LIN {X 0,Y 536.354,Z 685.03,A -85,B 0,C 180,E1 4123.665,E2 4123.665} C_VEL
LIN {X 0,Y 536.384,Z 685.03,A -85,B 0,C 180,E1 4128.647,E2 4128.647} C_VEL
LIN {X 0,Y 536.412,Z 685.03,A -85,B 0,C 180,E1 4133.543,E2 4133.543} C_VEL
LIN {X 0,Y 536.394,Z 685.03,A -85,B 0,C 180,E1 4138.392,E2 4138.392} C_VEL
LIN {X 0,Y 536.456,Z 685.03,A -85,B 0,C 180,E1 4143.228,E2 4143.228} C_VEL
LIN {X 0,Y 536.326,Z 685.03,A -85,B 0,C 180,E1 4148.09,E2 4148.09} C_VEL
LIN {X 0,Y 536.292,Z 685.03,A -85,B 0,C 180,E1 4153.011,E2 4153.011} C_VEL
LIN {X 0,Y 536.25,Z 685.03,A -85,B 0,C 180,E1 4158.034,E2 4158.034} C_VEL
LIN {X 0,Y 536.123,Z 685.03,A -85,B 0,C 180,E1 4163.209,E2 4163.209} C_VEL
LIN {X 0,Y 536.061,Z 685.03,A -85,B 0,C 180,E1 4166.771,E2 4166.771} C_VEL
LIN {X 0,Y 531.944,Z 685.03,A -85,B 0,C 180,E1 4168.601,E2 4168.601} C_VEL
LIN {X 0,Y 528.057,Z 685.03,A -85,B 0,C 180,E1 4170.459,E2 4170.459} C_VEL
LIN {X 0,Y 528.176,Z 685.03,A -85,B 0,C 180,E1 4176.874,E2 4176.874} C_VEL
LIN {X 0,Y 528.094,Z 685.03,A -85,B 0,C 180,E1 4183.298,E2 4183.298} C_VEL
LIN {X 0,Y 527.996,Z 685.03,A -85,B 0,C 180,E1 4188.904,E2 4188.904} C_VEL
LIN {X 0,Y 528.097,Z 685.034,A -85,B 0,C 180,E1 4193.319,E2 4193.319} C_VEL
LIN {X 0,Y 532.088,Z 694.126,A -85,B 0,C 180,E1 4194.343,E2 4194.343} C_VEL
LIN {X 0,Y 535.905,Z 698.294,A -85,B 0,C 180,E1 4195.482,E2 4195.482} C_VEL
LIN {X 0,Y 536.503,Z 702.972,A -85,B 0,C 180,E1 4195.991,E2 4195.991} C_VEL
LIN {X 0,Y 540.933,Z 714.461,A -85,B 0,C 180,E1 4196.486,E2 4196.486} C_VEL
LIN {X 0,Y 540.144,Z 776.912,A -85,B 0,C 180,E1 4197.563,E2 4197.563} C_VEL
LIN {X 0,Y 538.76,Z 815.29,A -85,B 0,C 180,E1 4198.857,E2 4198.857} C_VEL
LIN {X 0,Y 536.782,Z 852.451,A -85,B 0,C 180,E1 4200.764,E2 4200.764} C_VEL
LIN {X 0,Y 534.633,Z 888.686,A -85,B 0,C 180,E1 4203.381,E2 4203.381} C_VEL
LIN {X 0,Y 532.572,Z 920.102,A -85,B 0,C 180,E1 4206.409,E2 4206.409} C_VEL
LIN {X 0,Y 530.859,Z 948.755,A -85,B 0,C 180,E1 4210.057,E2 4210.057} C_VEL
LIN {X 0,Y 529.67,Z 971.396,A -85,B 0,C 180,E1 4213.874,E2 4213.874} C_VEL
LIN {X 0,Y 529.13,Z 988.021,A -85,B 0,C 180,E1 4217.652,E2 4217.652} C_VEL
LIN {X 0,Y 528.922,Z 999.717,A -85,B 0,C 180,E1 4221.388,E2 4221.388} C_VEL
LIN {X 0,Y 528.766,Z 1006.986,A -85,B 0,C 180,E1 4225.091,E2 4225.091} C_VEL
LIN {X 0,Y 528.757,Z 1010.108,A -85,B 0,C 180,E1 4228.367,E2 4228.367} C_VEL
LIN {X 0,Y 528.747,Z 1009.367,A -85,B 0,C 180,E1 4232.749,E2 4232.749} C_VEL
LIN {X 0,Y 528.862,Z 1004.239,A -85,B 0,C 180,E1 4236.556,E2 4236.556} C_VEL
LIN {X 0,Y 528.962,Z 994.396,A -85,B 0,C 180,E1 4240.488,E2 4240.488} C_VEL
LIN {X 0,Y 529.503,Z 979.171,A -85,B 0,C 180,E1 4244.506,E2 4244.506} C_VEL
LIN {X 0,Y 530.406,Z 958.359,A -85,B 0,C 180,E1 4248.455,E2 4248.455} C_VEL
LIN {X 0,Y 531.902,Z 931.392,A -85,B 0,C 180,E1 4252.271,E2 4252.271} C_VEL
LIN {X 0,Y 533.823,Z 900.632,A -85,B 0,C 180,E1 4255.566,E2 4255.566} C_VEL
LIN {X 0,Y 535.948,Z 866.542,A -85,B 0,C 180,E1 4258.318,E2 4258.318} C_VEL
LIN {X 0,Y 538.081,Z 828.372,A -85,B 0,C 180,E1 4260.553,E2 4260.553} C_VEL
LIN {X 0,Y 539.691,Z 789.324,A -85,B 0,C 180,E1 4262.095,E2 4262.095} C_VEL
LIN {X 0,Y 540.833,Z 748.246,A -85,B 0,C 180,E1 4262.995,E2 4262.995} C_VEL
LIN {X 0,Y 540.481,Z 711.306,A -85,B 0,C 180,E1 4263.595,E2 4263.595} C_VEL
LIN {X 0,Y 535.854,Z 701.121,A -85,B 0,C 180,E1 4264.154,E2 4264.154} C_VEL
LIN {X 0,Y 535.477,Z 697.832,A -85,B 0,C 180,E1 4264.694,E2 4264.694} C_VEL
LIN {X 0,Y 531.547,Z 693.051,A -85,B 0,C 180,E1 4265.81,E2 4265.81} C_VEL
LIN {X 0,Y 528.087,Z 685.03,A -85,B 0,C 180,E1 4266.686,E2 4266.686} C_VEL
LIN {X 0,Y 528.034,Z 685.03,A -85,B 0,C 180,E1 4273.31,E2 4273.31} C_VEL
LIN {X 0,Y 528.107,Z 685.03,A -85,B 0,C 180,E1 4278.913,E2 4278.913} C_VEL
LIN {X 0,Y 528.109,Z 685.03,A -85,B 0,C 180,E1 4285.146,E2 4285.146} C_VEL
LIN {X 0,Y 528.131,Z 685.03,A -85,B 0,C 180,E1 4290.938,E2 4290.938} C_VEL
LIN {X 0,Y 528.203,Z 685.03,A -85,B 0,C 180,E1 4296.422,E2 4296.422} C_VEL
LIN {X 0,Y 528.353,Z 685.03,A -85,B 0,C 180,E1 4302.243,E2 4302.243} C_VEL
LIN {X 0,Y 532.473,Z 702.678,A -85,B 0,C 180,E1 4302.729,E2 4302.729} C_VEL
LIN {X 0,Y 532.139,Z 746.804,A -85,B 0,C 180,E1 4303.524,E2 4303.524} C_VEL
LIN {X 0,Y 531.58,Z 774.498,A -85,B 0,C 180,E1 4304.67,E2 4304.67} C_VEL
LIN {X 0,Y 530.64,Z 800.027,A -85,B 0,C 180,E1 4306.429,E2 4306.429} C_VEL
LIN {X 0,Y 529.919,Z 821.879,A -85,B 0,C 180,E1 4308.72,E2 4308.72} C_VEL
LIN {X 0,Y 529.325,Z 840.1,A -85,B 0,C 180,E1 4311.596,E2 4311.596} C_VEL
LIN {X 0,Y 529.05,Z 851.376,A -85,B 0,C 180,E1 4314.267,E2 4314.267} C_VEL
LIN {X 0,Y 529.003,Z 857.801,A -85,B 0,C 180,E1 4316.844,E2 4316.844} C_VEL
LIN {X 0,Y 528.911,Z 860.413,A -85,B 0,C 180,E1 4319.996,E2 4319.996} C_VEL
LIN {X 0,Y 528.996,Z 857.464,A -85,B 0,C 180,E1 4323.267,E2 4323.267} C_VEL
LIN {X 0,Y 529.045,Z 849.615,A -85,B 0,C 180,E1 4326.136,E2 4326.136} C_VEL
LIN {X 0,Y 529.361,Z 835.063,A -85,B 0,C 180,E1 4329.223,E2 4329.223} C_VEL
LIN {X 0,Y 530.002,Z 817.359,A -85,B 0,C 180,E1 4331.7,E2 4331.7} C_VEL
LIN {X 0,Y 530.789,Z 794.591,A -85,B 0,C 180,E1 4333.874,E2 4333.874} C_VEL
LIN {X 0,Y 531.58,Z 768.365,A -85,B 0,C 180,E1 4335.503,E2 4335.503} C_VEL
LIN {X 0,Y 532.203,Z 738.767,A -85,B 0,C 180,E1 4336.565,E2 4336.565} C_VEL
LIN {X 0,Y 531.65,Z 697.002,A -85,B 0,C 180,E1 4337.27,E2 4337.27} C_VEL
LIN {X 0,Y 528.402,Z 685.03,A -85,B 0,C 180,E1 4337.66,E2 4337.66} C_VEL
LIN {X 0,Y 528.196,Z 685.03,A -85,B 0,C 180,E1 4343.894,E2 4343.894} C_VEL
LIN {X 0,Y 528.104,Z 685.03,A -85,B 0,C 180,E1 4349.055,E2 4349.055} C_VEL
LIN {X 0,Y 528.107,Z 685.03,A -85,B 0,C 180,E1 4354.845,E2 4354.845} C_VEL
LIN {X 0,Y 528.115,Z 685.03,A -85,B 0,C 180,E1 4359.505,E2 4359.505} C_VEL
LIN {X 0,Y 528.084,Z 685.03,A -85,B 0,C 180,E1 4365.582,E2 4365.582} C_VEL
LIN {X 0,Y 528.122,Z 685.03,A -85,B 0,C 180,E1 4371.047,E2 4371.047} C_VEL
LIN {X 0,Y 528.093,Z 685.03,A -85,B 0,C 180,E1 4377.113,E2 4377.113} C_VEL
LIN {X 0,Y 528.209,Z 685.03,A -85,B 0,C 180,E1 4382.796,E2 4382.796} C_VEL
LIN {X 0,Y 528.294,Z 685.296,A -85,B 0,C 180,E1 4386.535,E2 4386.535} C_VEL
LIN {X 0,Y 534.475,Z 708.657,A -85,B 0,C 180,E1 4387.48,E2 4387.48} C_VEL
LIN {X 0,Y 533.347,Z 740.861,A -85,B 0,C 180,E1 4388.886,E2 4388.886} C_VEL
LIN {X 0,Y 531.992,Z 771.472,A -85,B 0,C 180,E1 4390.958,E2 4390.958} C_VEL
LIN {X 0,Y 530.758,Z 798.135,A -85,B 0,C 180,E1 4393.479,E2 4393.479} C_VEL
LIN {X 0,Y 529.823,Z 820.92,A -85,B 0,C 180,E1 4396.46,E2 4396.46} C_VEL
LIN {X 0,Y 529.261,Z 838.534,A -85,B 0,C 180,E1 4399.708,E2 4399.708} C_VEL
LIN {X 0,Y 528.963,Z 850.704,A -85,B 0,C 180,E1 4403.033,E2 4403.033} C_VEL
LIN {X 0,Y 528.87,Z 858.388,A -85,B 0,C 180,E1 4406.726,E2 4406.726} C_VEL
LIN {X 0,Y 528.806,Z 860.497,A -85,B 0,C 180,E1 4409.998,E2 4409.998} C_VEL
LIN {X 0,Y 528.869,Z 858.264,A -85,B 0,C 180,E1 4413.269,E2 4413.269} C_VEL
LIN {X 0,Y 528.989,Z 850.471,A -85,B 0,C 180,E1 4416.961,E2 4416.961} C_VEL
LIN {X 0,Y 529.325,Z 837.086,A -85,B 0,C 180,E1 4420.514,E2 4420.514} C_VEL
LIN {X 0,Y 529.976,Z 817.91,A -85,B 0,C 180,E1 4423.9,E2 4423.9} C_VEL
LIN {X 0,Y 530.907,Z 793.972,A -85,B 0,C 180,E1 4426.887,E2 4426.887} C_VEL
LIN {X 0,Y 532.18,Z 766.335,A -85,B 0,C 180,E1 4429.352,E2 4429.352} C_VEL
LIN {X 0,Y 533.507,Z 736.298,A -85,B 0,C 180,E1 4431.263,E2 4431.263} C_VEL
LIN {X 0,Y 534.003,Z 703.097,A -85,B 0,C 180,E1 4432.636,E2 4432.636} C_VEL
LIN {X 0,Y 528.39,Z 685.03,A -85,B 0,C 180,E1 4433.406,E2 4433.406} C_VEL
LIN {X 0,Y 528.218,Z 685.03,A -85,B 0,C 180,E1 4439.054,E2 4439.054} C_VEL
LIN {X 0,Y 528.144,Z 685.03,A -85,B 0,C 180,E1 4444.849,E2 4444.849} C_VEL
LIN {X 0,Y 527.985,Z 685.03,A -85,B 0,C 180,E1 4451.097,E2 4451.097} C_VEL
LIN {X 0,Y 528.062,Z 685.03,A -85,B 0,C 180,E1 4456.709,E2 4456.709} C_VEL
LIN {X 0,Y 528.163,Z 685.03,A -85,B 0,C 180,E1 4463.128,E2 4463.128} C_VEL
LIN {X 0,Y 528.134,Z 685.03,A -85,B 0,C 180,E1 4469.056,E2 4469.056} C_VEL
LIN {X 0,Y 528.231,Z 685.03,A -85,B 0,C 180,E1 4474.634,E2 4474.634} C_VEL
LIN {X 0,Y 528.453,Z 685.03,A -85,B 0,C 180,E1 4480.445,E2 4480.445} C_VEL
LIN {X 0,Y 528.576,Z 685.03,A -85,B 0,C 180,E1 4486.803,E2 4486.803} C_VEL
LIN {X 0,Y 528.49,Z 685.03,A -85,B 0,C 180,E1 4492.655,E2 4492.655} C_VEL
LIN {X 0,Y 528.516,Z 685.03,A -85,B 0,C 180,E1 4498.368,E2 4498.368} C_VEL
LIN {X 0,Y 528.569,Z 685.03,A -85,B 0,C 180,E1 4503.277,E2 4503.277} C_VEL
LIN {X 0,Y 528.43,Z 685.03,A -85,B 0,C 180,E1 4508.212,E2 4508.212} C_VEL
LIN {X 0,Y 528.339,Z 685.03,A -85,B 0,C 180,E1 4513.811,E2 4513.811} C_VEL
LIN {X 0,Y 528.331,Z 685.03,A -85,B 0,C 180,E1 4519.517,E2 4519.517} C_VEL
LIN {X 0,Y 528.183,Z 685.03,A -85,B 0,C 180,E1 4525.377,E2 4525.377} C_VEL
LIN {X 0,Y 528.057,Z 685.03,A -85,B 0,C 180,E1 4530.459,E2 4530.459} C_VEL
LIN {X 0,Y 525.578,Z 685.03,A -85,B 0,C 180,E1 4531.861,E2 4531.861} C_VEL
LIN {X 0,Y 520.171,Z 685.03,A -85,B 0,C 180,E1 4533.962,E2 4533.962} C_VEL
LIN {X 0,Y 520.069,Z 685.03,A -85,B 0,C 180,E1 4534.205,E2 4534.205} C_VEL
LIN {X 0,Y 520.223,Z 685.03,A -85,B 0,C 180,E1 4539.655,E2 4539.655} C_VEL
LIN {X 0,Y 520.13,Z 685.03,A -85,B 0,C 180,E1 4545.871,E2 4545.871} C_VEL
LIN {X 0,Y 520.099,Z 685.03,A -85,B 0,C 180,E1 4551.57,E2 4551.57} C_VEL
LIN {X 0,Y 520.162,Z 685.3,A -85,B 0,C 180,E1 4552.811,E2 4552.811} C_VEL
LIN {X 0,Y 524.281,Z 695.521,A -85,B 0,C 180,E1 4553.697,E2 4553.697} C_VEL
LIN {X 0,Y 529.992,Z 703.357,A -85,B 0,C 180,E1 4554.791,E2 4554.791} C_VEL
LIN {X 0,Y 531.939,Z 706.912,A -85,B 0,C 180,E1 4555.435,E2 4555.435} C_VEL
LIN {X 0,Y 532.885,Z 711.836,A -85,B 0,C 180,E1 4555.869,E2 4555.869} C_VEL
LIN {X 0,Y 534.317,Z 717.12,A -85,B 0,C 180,E1 4556.057,E2 4556.057} C_VEL
LIN {X 0,Y 533.477,Z 776.899,A -85,B 0,C 180,E1 4557.107,E2 4557.107} C_VEL
LIN {X 0,Y 531.892,Z 815.592,A -85,B 0,C 180,E1 4558.424,E2 4558.424} C_VEL
LIN {X 0,Y 529.702,Z 853.612,A -85,B 0,C 180,E1 4560.413,E2 4560.413} C_VEL
LIN {X 0,Y 527.388,Z 888.681,A -85,B 0,C 180,E1 4562.986,E2 4562.986} C_VEL
LIN {X 0,Y 525.127,Z 920.219,A -85,B 0,C 180,E1 4566.068,E2 4566.068} C_VEL
LIN {X 0,Y 523.234,Z 948.76,A -85,B 0,C 180,E1 4569.754,E2 4569.754} C_VEL
LIN {X 0,Y 521.935,Z 971.4,A -85,B 0,C 180,E1 4573.629,E2 4573.629} C_VEL
LIN {X 0,Y 521.287,Z 988.024,A -85,B 0,C 180,E1 4577.463,E2 4577.463} C_VEL
LIN {X 0,Y 521.052,Z 999.717,A -85,B 0,C 180,E1 4581.257,E2 4581.257} C_VEL
LIN {X 0,Y 520.871,Z 1006.989,A -85,B 0,C 180,E1 4585.016,E2 4585.016} C_VEL
LIN {X 0,Y 520.87,Z 1010.11,A -85,B 0,C 180,E1 4588.342,E2 4588.342} C_VEL
LIN {X 0,Y 520.994,Z 1010.107,A -85,B 0,C 180,E1 4591.662,E2 4591.662} C_VEL
LIN {X 0,Y 520.997,Z 1005.741,A -85,B 0,C 180,E1 4595.821,E2 4595.821} C_VEL
LIN {X 0,Y 521.085,Z 996.126,A -85,B 0,C 180,E1 4600.075,E2 4600.075} C_VEL
LIN {X 0,Y 521.585,Z 981.334,A -85,B 0,C 180,E1 4604.23,E2 4604.23} C_VEL
LIN {X 0,Y 522.578,Z 961.26,A -85,B 0,C 180,E1 4608.245,E2 4608.245} C_VEL
LIN {X 0,Y 524.078,Z 936.283,A -85,B 0,C 180,E1 4611.986,E2 4611.986} C_VEL
LIN {X 0,Y 526.175,Z 905.44,A -85,B 0,C 180,E1 4615.483,E2 4615.483} C_VEL
LIN {X 0,Y 528.495,Z 871.136,A -85,B 0,C 180,E1 4618.404,E2 4618.404} C_VEL
LIN {X 0,Y 530.864,Z 833.862,A -85,B 0,C 180,E1 4620.715,E2 4620.715} C_VEL
LIN {X 0,Y 532.803,Z 795.147,A -85,B 0,C 180,E1 4622.354,E2 4622.354} C_VEL
LIN {X 0,Y 534.124,Z 756.8,A -85,B 0,C 180,E1 4623.314,E2 4623.314} C_VEL
LIN {X 0,Y 533.814,Z 713.846,A -85,B 0,C 180,E1 4624.031,E2 4624.031} C_VEL
LIN {X 0,Y 531.986,Z 709.074,A -85,B 0,C 180,E1 4624.335,E2 4624.335} C_VEL
LIN {X 0,Y 531.319,Z 704.389,A -85,B 0,C 180,E1 4624.917,E2 4624.917} C_VEL
LIN {X 0,Y 526.441,Z 699.138,A -85,B 0,C 180,E1 4625.909,E2 4625.909} C_VEL
LIN {X 0,Y 521.184,Z 689.298,A -85,B 0,C 180,E1 4626.821,E2 4626.821} C_VEL
LIN {X 0,Y 520.132,Z 685.03,A -85,B 0,C 180,E1 4627.142,E2 4627.142} C_VEL
LIN {X 0,Y 520.131,Z 685.03,A -85,B 0,C 180,E1 4633.506,E2 4633.506} C_VEL
LIN {X 0,Y 520.201,Z 685.03,A -85,B 0,C 180,E1 4638.964,E2 4638.964} C_VEL
LIN {X 0,Y 520.165,Z 685.03,A -85,B 0,C 180,E1 4644.534,E2 4644.534} C_VEL
LIN {X 0,Y 520.203,Z 685.03,A -85,B 0,C 180,E1 4650.497,E2 4650.497} C_VEL
LIN {X 0,Y 520.302,Z 685.03,A -85,B 0,C 180,E1 4656.042,E2 4656.042} C_VEL
LIN {X 0,Y 520.458,Z 685.03,A -85,B 0,C 180,E1 4661.896,E2 4661.896} C_VEL
LIN {X 0,Y 525.118,Z 704.487,A -85,B 0,C 180,E1 4662.445,E2 4662.445} C_VEL
LIN {X 0,Y 524.688,Z 748.901,A -85,B 0,C 180,E1 4663.283,E2 4663.283} C_VEL
LIN {X 0,Y 524.081,Z 776.919,A -85,B 0,C 180,E1 4664.484,E2 4664.484} C_VEL
LIN {X 0,Y 523.141,Z 801.802,A -85,B 0,C 180,E1 4666.242,E2 4666.242} C_VEL
LIN {X 0,Y 522.363,Z 823.118,A -85,B 0,C 180,E1 4668.512,E2 4668.512} C_VEL
LIN {X 0,Y 521.688,Z 840.432,A -85,B 0,C 180,E1 4671.262,E2 4671.262} C_VEL
LIN {X 0,Y 521.247,Z 852.269,A -85,B 0,C 180,E1 4674.181,E2 4674.181} C_VEL
LIN {X 0,Y 521.09,Z 859.131,A -85,B 0,C 180,E1 4677.362,E2 4677.362} C_VEL
LIN {X 0,Y 521.032,Z 860.825,A -85,B 0,C 180,E1 4679.996,E2 4679.996} C_VEL
LIN {X 0,Y 521.117,Z 857.949,A -85,B 0,C 180,E1 4683.316,E2 4683.316} C_VEL
LIN {X 0,Y 521.262,Z 848.872,A -85,B 0,C 180,E1 4686.645,E2 4686.645} C_VEL
LIN {X 0,Y 521.691,Z 834.958,A -85,B 0,C 180,E1 4689.569,E2 4689.569} C_VEL
LIN {X 0,Y 522.477,Z 814.795,A -85,B 0,C 180,E1 4692.294,E2 4692.294} C_VEL
LIN {X 0,Y 523.284,Z 791.675,A -85,B 0,C 180,E1 4694.381,E2 4694.381} C_VEL
LIN {X 0,Y 524.182,Z 764.331,A -85,B 0,C 180,E1 4695.974,E2 4695.974} C_VEL
LIN {X 0,Y 524.733,Z 735.414,A -85,B 0,C 180,E1 4696.912,E2 4696.912} C_VEL
LIN {X 0,Y 524.25,Z 698.598,A -85,B 0,C 180,E1 4697.53,E2 4697.53} C_VEL
LIN {X 0,Y 520.493,Z 685.03,A -85,B 0,C 180,E1 4697.928,E2 4697.928} C_VEL
LIN {X 0,Y 520.3,Z 685.03,A -85,B 0,C 180,E1 4703.95,E2 4703.95} C_VEL
LIN {X 0,Y 520.176,Z 685.03,A -85,B 0,C 180,E1 4709.541,E2 4709.541} C_VEL
LIN {X 0,Y 520.204,Z 685.03,A -85,B 0,C 180,E1 4715.678,E2 4715.678} C_VEL
LIN {X 0,Y 520.144,Z 685.03,A -85,B 0,C 180,E1 4721.029,E2 4721.029} C_VEL
LIN {X 0,Y 520.167,Z 685.03,A -85,B 0,C 180,E1 4726.479,E2 4726.479} C_VEL
LIN {X 0,Y 520.207,Z 685.03,A -85,B 0,C 180,E1 4732.466,E2 4732.466} C_VEL
LIN {X 0,Y 520.218,Z 685.03,A -85,B 0,C 180,E1 4738.52,E2 4738.52} C_VEL
LIN {X 0,Y 520.312,Z 685.03,A -85,B 0,C 180,E1 4744.209,E2 4744.209} C_VEL
LIN {X 0,Y 520.395,Z 685.6,A -85,B 0,C 180,E1 4746.14,E2 4746.14} C_VEL
LIN {X 0,Y 527.258,Z 710.651,A -85,B 0,C 180,E1 4747.185,E2 4747.185} C_VEL
LIN {X 0,Y 526.023,Z 743.222,A -85,B 0,C 180,E1 4748.647,E2 4748.647} C_VEL
LIN {X 0,Y 524.583,Z 772.51,A -85,B 0,C 180,E1 4750.679,E2 4750.679} C_VEL
LIN {X 0,Y 523.113,Z 798.31,A -85,B 0,C 180,E1 4753.23,E2 4753.23} C_VEL
LIN {X 0,Y 521.98,Z 822.179,A -85,B 0,C 180,E1 4756.46,E2 4756.46} C_VEL
LIN {X 0,Y 521.407,Z 839.142,A -85,B 0,C 180,E1 4759.687,E2 4759.687} C_VEL
LIN {X 0,Y 521.027,Z 851.834,A -85,B 0,C 180,E1 4763.345,E2 4763.345} C_VEL
LIN {X 0,Y 520.97,Z 858.387,A -85,B 0,C 180,E1 4766.676,E2 4766.676} C_VEL
LIN {X 0,Y 520.91,Z 860.497,A -85,B 0,C 180,E1 4769.997,E2 4769.997} C_VEL
LIN {X 0,Y 520.969,Z 858.265,A -85,B 0,C 180,E1 4773.319,E2 4773.319} C_VEL
LIN {X 0,Y 521.127,Z 850.474,A -85,B 0,C 180,E1 4777.067,E2 4777.067} C_VEL
LIN {X 0,Y 521.439,Z 837.884,A -85,B 0,C 180,E1 4780.499,E2 4780.499} C_VEL
LIN {X 0,Y 522.128,Z 819.589,A -85,B 0,C 180,E1 4783.864,E2 4783.864} C_VEL
LIN {X 0,Y 523.275,Z 794.687,A -85,B 0,C 180,E1 4787.1,E2 4787.1} C_VEL
LIN {X 0,Y 524.821,Z 767.548,A -85,B 0,C 180,E1 4789.635,E2 4789.635} C_VEL
LIN {X 0,Y 526.274,Z 737.203,A -85,B 0,C 180,E1 4791.587,E2 4791.587} C_VEL
LIN {X 0,Y 526.687,Z 704.594,A -85,B 0,C 180,E1 4792.96,E2 4792.96} C_VEL
LIN {X 0,Y 520.413,Z 685.03,A -85,B 0,C 180,E1 4793.815,E2 4793.815} C_VEL
LIN {X 0,Y 520.264,Z 685.03,A -85,B 0,C 180,E1 4799.542,E2 4799.542} C_VEL
LIN {X 0,Y 520.158,Z 685.03,A -85,B 0,C 180,E1 4805.464,E2 4805.464} C_VEL
LIN {X 0,Y 520.075,Z 685.03,A -85,B 0,C 180,E1 4811.862,E2 4811.862} C_VEL
LIN {X 0,Y 520.172,Z 685.03,A -85,B 0,C 180,E1 4818.156,E2 4818.156} C_VEL
LIN {X 0,Y 520.189,Z 685.03,A -85,B 0,C 180,E1 4824.316,E2 4824.316} C_VEL
LIN {X 0,Y 520.227,Z 685.03,A -85,B 0,C 180,E1 4830.482,E2 4830.482} C_VEL
LIN {X 0,Y 520.314,Z 685.03,A -85,B 0,C 180,E1 4836.051,E2 4836.051} C_VEL
LIN {X 0,Y 520.508,Z 685.03,A -85,B 0,C 180,E1 4841.409,E2 4841.409} C_VEL
LIN {X 0,Y 520.681,Z 685.03,A -85,B 0,C 180,E1 4846.599,E2 4846.599} C_VEL
LIN {X 0,Y 520.575,Z 685.03,A -85,B 0,C 180,E1 4852.656,E2 4852.656} C_VEL
LIN {X 0,Y 520.641,Z 685.03,A -85,B 0,C 180,E1 4858.343,E2 4858.343} C_VEL
LIN {X 0,Y 520.664,Z 685.03,A -85,B 0,C 180,E1 4863.326,E2 4863.326} C_VEL
LIN {X 0,Y 520.518,Z 685.03,A -85,B 0,C 180,E1 4868.338,E2 4868.338} C_VEL
LIN {X 0,Y 520.48,Z 685.03,A -85,B 0,C 180,E1 4873.414,E2 4873.414} C_VEL
LIN {X 0,Y 520.416,Z 685.03,A -85,B 0,C 180,E1 4878.602,E2 4878.602} C_VEL
LIN {X 0,Y 520.272,Z 685.03,A -85,B 0,C 180,E1 4883.959,E2 4883.959} C_VEL
LIN {X 0,Y 520.174,Z 685.03,A -85,B 0,C 180,E1 4889.55,E2 4889.55} C_VEL
LIN {X 0,Y 520.069,Z 685.03,A -85,B 0,C 180,E1 4894.205,E2 4894.205} C_VEL
LIN {X 0,Y 516.137,Z 685.03,A -85,B 0,C 180,E1 4896.091,E2 4896.091} C_VEL
LIN {X 0,Y 512.287,Z 685.03,A -85,B 0,C 180,E1 4898.006,E2 4898.006} C_VEL
LIN {X 0,Y 512.255,Z 685.03,A -85,B 0,C 180,E1 4902.652,E2 4902.652} C_VEL
LIN {X 0,Y 512.163,Z 685.03,A -85,B 0,C 180,E1 4907.441,E2 4907.441} C_VEL
LIN {X 0,Y 512.192,Z 685.146,A -85,B 0,C 180,E1 4912.26,E2 4912.26} C_VEL
LIN {X 0,Y 517.631,Z 699.651,A -85,B 0,C 180,E1 4913.517,E2 4913.517} C_VEL
LIN {X 0,Y 524.978,Z 709.353,A -85,B 0,C 180,E1 4914.648,E2 4914.648} C_VEL
LIN {X 0,Y 527.259,Z 714.744,A -85,B 0,C 180,E1 4915.325,E2 4915.325} C_VEL
LIN {X 0,Y 527.77,Z 718.696,A -85,B 0,C 180,E1 4915.603,E2 4915.603} C_VEL
LIN {X 0,Y 526.841,Z 777.247,A -85,B 0,C 180,E1 4916.649,E2 4916.649} C_VEL
LIN {X 0,Y 525.111,Z 815.585,A -85,B 0,C 180,E1 4917.968,E2 4917.968} C_VEL
LIN {X 0,Y 522.754,Z 852.996,A -85,B 0,C 180,E1 4919.938,E2 4919.938} C_VEL
LIN {X 0,Y 520.179,Z 888.679,A -85,B 0,C 180,E1 4922.581,E2 4922.581} C_VEL
LIN {X 0,Y 517.707,Z 920.398,A -85,B 0,C 180,E1 4925.724,E2 4925.724} C_VEL
LIN {X 0,Y 515.594,Z 949.007,A -85,B 0,C 180,E1 4929.478,E2 4929.478} C_VEL
LIN {X 0,Y 514.187,Z 971.403,A -85,B 0,C 180,E1 4933.375,E2 4933.375} C_VEL
LIN {X 0,Y 513.478,Z 988.028,A -85,B 0,C 180,E1 4937.269,E2 4937.269} C_VEL
LIN {X 0,Y 513.156,Z 1000.722,A -85,B 0,C 180,E1 4941.547,E2 4941.547} C_VEL
LIN {X 0,Y 512.979,Z 1006.991,A -85,B 0,C 180,E1 4944.939,E2 4944.939} C_VEL
LIN {X 0,Y 512.993,Z 1010.111,A -85,B 0,C 180,E1 4948.317,E2 4948.317} C_VEL
LIN {X 0,Y 513.109,Z 1010.108,A -85,B 0,C 180,E1 4951.688,E2 4951.688} C_VEL
LIN {X 0,Y 513.102,Z 1005.74,A -85,B 0,C 180,E1 4955.911,E2 4955.911} C_VEL
LIN {X 0,Y 513.214,Z 996.317,A -85,B 0,C 180,E1 4960.164,E2 4960.164} C_VEL
LIN {X 0,Y 513.739,Z 982.207,A -85,B 0,C 180,E1 4964.237,E2 4964.237} C_VEL
LIN {X 0,Y 514.816,Z 962.388,A -85,B 0,C 180,E1 4968.326,E2 4968.326} C_VEL
LIN {X 0,Y 516.523,Z 936.281,A -85,B 0,C 180,E1 4972.325,E2 4972.325} C_VEL
LIN {X 0,Y 518.822,Z 905.439,A -85,B 0,C 180,E1 4975.871,E2 4975.871} C_VEL
LIN {X 0,Y 521.365,Z 871.904,A -85,B 0,C 180,E1 4978.767,E2 4978.767} C_VEL
LIN {X 0,Y 523.942,Z 834.623,A -85,B 0,C 180,E1 4981.122,E2 4981.122} C_VEL
LIN {X 0,Y 526.056,Z 795.898,A -85,B 0,C 180,E1 4982.793,E2 4982.793} C_VEL
LIN {X 0,Y 527.517,Z 757.791,A -85,B 0,C 180,E1 4983.769,E2 4983.769} C_VEL
LIN {X 0,Y 527.562,Z 716.814,A -85,B 0,C 180,E1 4984.456,E2 4984.456} C_VEL
LIN {X 0,Y 526.094,Z 710.29,A -85,B 0,C 180,E1 4985.167,E2 4985.167} C_VEL
LIN {X 0,Y 519.052,Z 701.862,A -85,B 0,C 180,E1 4986.228,E2 4986.228} C_VEL
LIN {X 0,Y 513.064,Z 689.146,A -85,B 0,C 180,E1 4987.202,E2 4987.202} C_VEL
LIN {X 0,Y 512.175,Z 685.03,A -85,B 0,C 180,E1 4987.553,E2 4987.553} C_VEL
LIN {X 0,Y 512.187,Z 685.03,A -85,B 0,C 180,E1 4992.665,E2 4992.665} C_VEL
LIN {X 0,Y 512.26,Z 685.03,A -85,B 0,C 180,E1 4997.436,E2 4997.436} C_VEL
LIN {X 0,Y 512.269,Z 685.03,A -85,B 0,C 180,E1 5002.696,E2 5002.696} C_VEL
LIN {X 0,Y 512.257,Z 685.03,A -85,B 0,C 180,E1 5008.69,E2 5008.69} C_VEL
LIN {X 0,Y 512.327,Z 685.03,A -85,B 0,C 180,E1 5013.779,E2 5013.779} C_VEL
LIN {X 0,Y 512.462,Z 685.03,A -85,B 0,C 180,E1 5019.305,E2 5019.305} C_VEL
LIN {X 0,Y 512.549,Z 685.552,A -85,B 0,C 180,E1 5021.537,E2 5021.537} C_VEL
LIN {X 0,Y 517.769,Z 703.512,A -85,B 0,C 180,E1 5022.11,E2 5022.11} C_VEL
LIN {X 0,Y 517.288,Z 750.923,A -85,B 0,C 180,E1 5023.037,E2 5023.037} C_VEL
LIN {X 0,Y 516.669,Z 778,A -85,B 0,C 180,E1 5024.216,E2 5024.216} C_VEL
LIN {X 0,Y 515.642,Z 803.277,A -85,B 0,C 180,E1 5026.026,E2 5026.026} C_VEL
LIN {X 0,Y 514.745,Z 825.334,A -85,B 0,C 180,E1 5028.429,E2 5028.429} C_VEL
LIN {X 0,Y 513.975,Z 843.001,A -85,B 0,C 180,E1 5031.343,E2 5031.343} C_VEL
LIN {X 0,Y 513.471,Z 854.905,A -85,B 0,C 180,E1 5034.516,E2 5034.516} C_VEL
LIN {X 0,Y 513.333,Z 860.727,A -85,B 0,C 180,E1 5037.469,E2 5037.469} C_VEL
LIN {X 0,Y 513.282,Z 862.188,A -85,B 0,C 180,E1 5039.996,E2 5039.996} C_VEL
LIN {X 0,Y 513.352,Z 859.214,A -85,B 0,C 180,E1 5043.366,E2 5043.366} C_VEL
LIN {X 0,Y 513.51,Z 850.089,A -85,B 0,C 180,E1 5046.746,E2 5046.746} C_VEL
LIN {X 0,Y 513.996,Z 836.089,A -85,B 0,C 180,E1 5049.714,E2 5049.714} C_VEL
LIN {X 0,Y 514.857,Z 815.868,A -85,B 0,C 180,E1 5052.478,E2 5052.478} C_VEL
LIN {X 0,Y 515.729,Z 792.128,A -85,B 0,C 180,E1 5054.64,E2 5054.64} C_VEL
LIN {X 0,Y 516.695,Z 764.192,A -85,B 0,C 180,E1 5056.266,E2 5056.266} C_VEL
LIN {X 0,Y 517.273,Z 734.612,A -85,B 0,C 180,E1 5057.205,E2 5057.205} C_VEL
LIN {X 0,Y 516.63,Z 699.556,A -85,B 0,C 180,E1 5057.803,E2 5057.803} C_VEL
LIN {X 0,Y 512.554,Z 685.03,A -85,B 0,C 180,E1 5058.248,E2 5058.248} C_VEL
LIN {X 0,Y 512.359,Z 685.03,A -85,B 0,C 180,E1 5064.345,E2 5064.345} C_VEL
LIN {X 0,Y 512.213,Z 685.03,A -85,B 0,C 180,E1 5070.048,E2 5070.048} C_VEL
LIN {X 0,Y 512.286,Z 685.03,A -85,B 0,C 180,E1 5076.087,E2 5076.087} C_VEL
LIN {X 0,Y 512.257,Z 685.03,A -85,B 0,C 180,E1 5080.387,E2 5080.387} C_VEL
LIN {X 0,Y 512.206,Z 685.03,A -85,B 0,C 180,E1 5084.997,E2 5084.997} C_VEL
LIN {X 0,Y 512.288,Z 685.03,A -85,B 0,C 180,E1 5089.972,E2 5089.972} C_VEL
LIN {X 0,Y 512.194,Z 685.03,A -85,B 0,C 180,E1 5095.955,E2 5095.955} C_VEL
LIN {X 0,Y 512.36,Z 685.03,A -85,B 0,C 180,E1 5102.057,E2 5102.057} C_VEL
LIN {X 0,Y 512.427,Z 685.062,A -85,B 0,C 180,E1 5105.711,E2 5105.711} C_VEL
LIN {X 0,Y 520.066,Z 712.731,A -85,B 0,C 180,E1 5106.885,E2 5106.885} C_VEL
LIN {X 0,Y 518.771,Z 744.492,A -85,B 0,C 180,E1 5108.337,E2 5108.337} C_VEL
LIN {X 0,Y 517.221,Z 773.73,A -85,B 0,C 180,E1 5110.392,E2 5110.392} C_VEL
LIN {X 0,Y 515.627,Z 799.545,A -85,B 0,C 180,E1 5112.98,E2 5112.98} C_VEL
LIN {X 0,Y 514.318,Z 822.023,A -85,B 0,C 180,E1 5116.151,E2 5116.151} C_VEL
LIN {X 0,Y 513.471,Z 840.437,A -85,B 0,C 180,E1 5119.841,E2 5119.841} C_VEL
LIN {X 0,Y 513.165,Z 851.831,A -85,B 0,C 180,E1 5123.242,E2 5123.242} C_VEL
LIN {X 0,Y 513.081,Z 858.387,A -85,B 0,C 180,E1 5126.625,E2 5126.625} C_VEL
LIN {X 0,Y 512.993,Z 860.423,A -85,B 0,C 180,E1 5130.376,E2 5130.376} C_VEL
LIN {X 0,Y 513.103,Z 857.062,A -85,B 0,C 180,E1 5134.214,E2 5134.214} C_VEL
LIN {X 0,Y 513.335,Z 847.901,A -85,B 0,C 180,E1 5138.024,E2 5138.024} C_VEL
LIN {X 0,Y 513.801,Z 833.266,A -85,B 0,C 180,E1 5141.647,E2 5141.647} C_VEL
LIN {X 0,Y 514.819,Z 813.602,A -85,B 0,C 180,E1 5145.081,E2 5145.081} C_VEL
LIN {X 0,Y 516.236,Z 789.868,A -85,B 0,C 180,E1 5148.011,E2 5148.011} C_VEL
LIN {X 0,Y 517.896,Z 761.609,A -85,B 0,C 180,E1 5150.464,E2 5150.464} C_VEL
LIN {X 0,Y 519.3,Z 731.077,A -85,B 0,C 180,E1 5152.274,E2 5152.274} C_VEL
LIN {X 0,Y 519.362,Z 706.232,A -85,B 0,C 180,E1 5153.289,E2 5153.289} C_VEL
LIN {X 0,Y 512.459,Z 685.03,A -85,B 0,C 180,E1 5154.256,E2 5154.256} C_VEL
LIN {X 0,Y 512.3,Z 685.03,A -85,B 0,C 180,E1 5160.048,E2 5160.048} C_VEL
LIN {X 0,Y 512.201,Z 685.03,A -85,B 0,C 180,E1 5166.101,E2 5166.101} C_VEL
LIN {X 0,Y 512.178,Z 685.03,A -85,B 0,C 180,E1 5170.403,E2 5170.403} C_VEL
LIN {X 0,Y 512.173,Z 685.03,A -85,B 0,C 180,E1 5175.01,E2 5175.01} C_VEL
LIN {X 0,Y 512.296,Z 685.03,A -85,B 0,C 180,E1 5179.982,E2 5179.982} C_VEL
LIN {X 0,Y 512.232,Z 685.03,A -85,B 0,C 180,E1 5185.971,E2 5185.971} C_VEL
LIN {X 0,Y 512.328,Z 685.03,A -85,B 0,C 180,E1 5192.082,E2 5192.082} C_VEL
LIN {X 0,Y 512.428,Z 685.03,A -85,B 0,C 180,E1 5197.497,E2 5197.497} C_VEL
LIN {X 0,Y 512.639,Z 685.03,A -85,B 0,C 180,E1 5202.886,E2 5202.886} C_VEL
LIN {X 0,Y 512.668,Z 685.03,A -85,B 0,C 180,E1 5208.114,E2 5208.114} C_VEL
LIN {X 0,Y 512.705,Z 685.03,A -85,B 0,C 180,E1 5213.243,E2 5213.243} C_VEL
LIN {X 0,Y 512.741,Z 685.03,A -85,B 0,C 180,E1 5218.317,E2 5218.317} C_VEL
LIN {X 0,Y 512.769,Z 685.03,A -85,B 0,C 180,E1 5223.378,E2 5223.378} C_VEL
LIN {X 0,Y 512.611,Z 685.03,A -85,B 0,C 180,E1 5228.467,E2 5228.467} C_VEL
LIN {X 0,Y 512.542,Z 685.03,A -85,B 0,C 180,E1 5233.693,E2 5233.693} C_VEL
LIN {X 0,Y 512.469,Z 685.03,A -85,B 0,C 180,E1 5239.564,E2 5239.564} C_VEL
LIN {X 0,Y 512.335,Z 685.03,A -85,B 0,C 180,E1 5244.354,E2 5244.354} C_VEL
LIN {X 0,Y 512.211,Z 685.03,A -85,B 0,C 180,E1 5250.056,E2 5250.056} C_VEL
LIN {X 0,Y 512.251,Z 685.03,A -85,B 0,C 180,E1 5256.099,E2 5256.099} C_VEL
LIN {X 0,Y 512.287,Z 685.03,A -85,B 0,C 180,E1 5258.006,E2 5258.006} C_VEL
LIN {X 0,Y 509.808,Z 685.03,A -85,B 0,C 180,E1 5259.436,E2 5259.436} C_VEL
LIN {X 0,Y 504.243,Z 685.03,A -85,B 0,C 180,E1 5261.826,E2 5261.826} C_VEL
LIN {X 0,Y 504.187,Z 685.03,A -85,B 0,C 180,E1 5266.499,E2 5266.499} C_VEL
LIN {X 0,Y 504.322,Z 685.713,A -85,B 0,C 180,E1 5271.742,E2 5271.742} C_VEL
LIN {X 0,Y 511.317,Z 704.209,A -85,B 0,C 180,E1 5273.381,E2 5273.381} C_VEL
LIN {X 0,Y 521.17,Z 717.935,A -85,B 0,C 180,E1 5274.88,E2 5274.88} C_VEL
LIN {X 0,Y 521.178,Z 724.456,A -85,B 0,C 180,E1 5275.2,E2 5275.2} C_VEL
LIN {X 0,Y 520.179,Z 778.605,A -85,B 0,C 180,E1 5276.204,E2 5276.204} C_VEL
LIN {X 0,Y 518.33,Z 816.283,A -85,B 0,C 180,E1 5277.532,E2 5277.532} C_VEL
LIN {X 0,Y 515.728,Z 854.016,A -85,B 0,C 180,E1 5279.556,E2 5279.556} C_VEL
LIN {X 0,Y 512.883,Z 889.667,A -85,B 0,C 180,E1 5282.249,E2 5282.249} C_VEL
LIN {X 0,Y 510.163,Z 922.025,A -85,B 0,C 180,E1 5285.539,E2 5285.539} C_VEL
LIN {X 0,Y 507.905,Z 950.005,A -85,B 0,C 180,E1 5289.31,E2 5289.31} C_VEL
LIN {X 0,Y 506.363,Z 972.478,A -85,B 0,C 180,E1 5293.333,E2 5293.333} C_VEL
LIN {X 0,Y 505.56,Z 989.569,A -85,B 0,C 180,E1 5297.504,E2 5297.504} C_VEL
LIN {X 0,Y 505.264,Z 1000.725,A -85,B 0,C 180,E1 5301.414,E2 5301.414} C_VEL
LIN {X 0,Y 505.087,Z 1006.994,A -85,B 0,C 180,E1 5304.86,E2 5304.86} C_VEL
LIN {X 0,Y 505.09,Z 1010.112,A -85,B 0,C 180,E1 5308.291,E2 5308.291} C_VEL
LIN {X 0,Y 505.202,Z 1010.11,A -85,B 0,C 180,E1 5311.714,E2 5311.714} C_VEL
LIN {X 0,Y 505.211,Z 1005.739,A -85,B 0,C 180,E1 5316.004,E2 5316.004} C_VEL
LIN {X 0,Y 505.331,Z 996.316,A -85,B 0,C 180,E1 5320.325,E2 5320.325} C_VEL
LIN {X 0,Y 505.99,Z 981.087,A -85,B 0,C 180,E1 5324.737,E2 5324.737} C_VEL
LIN {X 0,Y 507.172,Z 960.892,A -85,B 0,C 180,E1 5328.885,E2 5328.885} C_VEL
LIN {X 0,Y 509.119,Z 934.459,A -85,B 0,C 180,E1 5332.916,E2 5332.916} C_VEL
LIN {X 0,Y 511.756,Z 903.197,A -85,B 0,C 180,E1 5336.491,E2 5336.491} C_VEL
LIN {X 0,Y 514.52,Z 868.916,A -85,B 0,C 180,E1 5339.427,E2 5339.427} C_VEL
LIN {X 0,Y 517.352,Z 831.713,A -85,B 0,C 180,E1 5341.734,E2 5341.734} C_VEL
LIN {X 0,Y 519.544,Z 792.025,A -85,B 0,C 180,E1 5343.405,E2 5343.405} C_VEL
LIN {X 0,Y 521.064,Z 750.75,A -85,B 0,C 180,E1 5344.377,E2 5344.377} C_VEL
LIN {X 0,Y 521.662,Z 719.901,A -85,B 0,C 180,E1 5344.943,E2 5344.943} C_VEL
LIN {X 0,Y 520.263,Z 715.673,A -85,B 0,C 180,E1 5345.338,E2 5345.338} C_VEL
LIN {X 0,Y 509.915,Z 702.399,A -85,B 0,C 180,E1 5346.61,E2 5346.61} C_VEL
LIN {X 0,Y 504.279,Z 685.03,A -85,B 0,C 180,E1 5347.87,E2 5347.87} C_VEL
LIN {X 0,Y 504.238,Z 685.03,A -85,B 0,C 180,E1 5354.091,E2 5354.091} C_VEL
LIN {X 0,Y 504.299,Z 685.03,A -85,B 0,C 180,E1 5358.829,E2 5358.829} C_VEL
LIN {X 0,Y 504.375,Z 685.03,A -85,B 0,C 180,E1 5363.889,E2 5363.889} C_VEL
LIN {X 0,Y 504.304,Z 685.03,A -85,B 0,C 180,E1 5370.209,E2 5370.209} C_VEL
LIN {X 0,Y 504.413,Z 685.03,A -85,B 0,C 180,E1 5375.238,E2 5375.238} C_VEL
LIN {X 0,Y 504.575,Z 685.031,A -85,B 0,C 180,E1 5381.118,E2 5381.118} C_VEL
LIN {X 0,Y 510.438,Z 706.142,A -85,B 0,C 180,E1 5381.824,E2 5381.824} C_VEL
LIN {X 0,Y 509.868,Z 752.872,A -85,B 0,C 180,E1 5382.783,E2 5382.783} C_VEL
LIN {X 0,Y 509.221,Z 779.689,A -85,B 0,C 180,E1 5383.978,E2 5383.978} C_VEL
LIN {X 0,Y 508.191,Z 803.574,A -85,B 0,C 180,E1 5385.696,E2 5385.696} C_VEL
LIN {X 0,Y 507.278,Z 824.775,A -85,B 0,C 180,E1 5387.979,E2 5387.979} C_VEL
LIN {X 0,Y 506.431,Z 842.357,A -85,B 0,C 180,E1 5390.781,E2 5390.781} C_VEL
LIN {X 0,Y 505.804,Z 855.149,A -85,B 0,C 180,E1 5394.003,E2 5394.003} C_VEL
LIN {X 0,Y 505.589,Z 862.124,A -85,B 0,C 180,E1 5397.43,E2 5397.43} C_VEL
LIN {X 0,Y 505.528,Z 863.551,A -85,B 0,C 180,E1 5399.996,E2 5399.996} C_VEL
LIN {X 0,Y 505.595,Z 860.478,A -85,B 0,C 180,E1 5403.418,E2 5403.418} C_VEL
LIN {X 0,Y 505.77,Z 851.305,A -85,B 0,C 180,E1 5406.85,E2 5406.85} C_VEL
LIN {X 0,Y 506.294,Z 837.22,A -85,B 0,C 180,E1 5409.863,E2 5409.863} C_VEL
LIN {X 0,Y 507.159,Z 818.821,A -85,B 0,C 180,E1 5412.453,E2 5412.453} C_VEL
LIN {X 0,Y 508.132,Z 795.272,A -85,B 0,C 180,E1 5414.703,E2 5414.703} C_VEL
LIN {X 0,Y 509.086,Z 768.748,A -85,B 0,C 180,E1 5416.35,E2 5416.35} C_VEL
LIN {X 0,Y 509.751,Z 739.215,A -85,B 0,C 180,E1 5417.393,E2 5417.393} C_VEL
LIN {X 0,Y 509.252,Z 701.263,A -85,B 0,C 180,E1 5418.064,E2 5418.064} C_VEL
LIN {X 0,Y 504.625,Z 685.03,A -85,B 0,C 180,E1 5418.595,E2 5418.595} C_VEL
LIN {X 0,Y 504.401,Z 685.03,A -85,B 0,C 180,E1 5424.754,E2 5424.754} C_VEL
LIN {X 0,Y 504.303,Z 685.03,A -85,B 0,C 180,E1 5430.569,E2 5430.569} C_VEL
LIN {X 0,Y 504.408,Z 685.03,A -85,B 0,C 180,E1 5436.742,E2 5436.742} C_VEL
LIN {X 0,Y 504.225,Z 685.03,A -85,B 0,C 180,E1 5441.56,E2 5441.56} C_VEL
LIN {X 0,Y 504.229,Z 685.03,A -85,B 0,C 180,E1 5446.496,E2 5446.496} C_VEL
LIN {X 0,Y 504.367,Z 685.03,A -85,B 0,C 180,E1 5453.241,E2 5453.241} C_VEL
LIN {X 0,Y 504.38,Z 685.03,A -85,B 0,C 180,E1 5459.424,E2 5459.424} C_VEL
LIN {X 0,Y 504.485,Z 685.03,A -85,B 0,C 180,E1 5465.276,E2 5465.276} C_VEL
LIN {X 0,Y 512.906,Z 713.471,A -85,B 0,C 180,E1 5466.528,E2 5466.528} C_VEL
LIN {X 0,Y 511.563,Z 745.118,A -85,B 0,C 180,E1 5467.981,E2 5467.981} C_VEL
LIN {X 0,Y 509.902,Z 774.942,A -85,B 0,C 180,E1 5470.099,E2 5470.099} C_VEL
LIN {X 0,Y 508.154,Z 800.777,A -85,B 0,C 180,E1 5472.721,E2 5472.721} C_VEL
LIN {X 0,Y 506.803,Z 822.317,A -85,B 0,C 180,E1 5475.774,E2 5475.774} C_VEL
LIN {X 0,Y 505.814,Z 839.52,A -85,B 0,C 180,E1 5479.251,E2 5479.251} C_VEL
LIN {X 0,Y 505.411,Z 850.918,A -85,B 0,C 180,E1 5482.707,E2 5482.707} C_VEL
LIN {X 0,Y 505.18,Z 858.386,A -85,B 0,C 180,E1 5486.572,E2 5486.572} C_VEL
LIN {X 0,Y 505.16,Z 860.498,A -85,B 0,C 180,E1 5489.997,E2 5489.997} C_VEL
LIN {X 0,Y 505.179,Z 858.267,A -85,B 0,C 180,E1 5493.423,E2 5493.423} C_VEL
LIN {X 0,Y 505.481,Z 849.519,A -85,B 0,C 180,E1 5497.718,E2 5497.718} C_VEL
LIN {X 0,Y 506.083,Z 835.436,A -85,B 0,C 180,E1 5501.609,E2 5501.609} C_VEL
LIN {X 0,Y 507.183,Z 816.554,A -85,B 0,C 180,E1 5505.059,E2 5505.059} C_VEL
LIN {X 0,Y 508.738,Z 792.295,A -85,B 0,C 180,E1 5508.153,E2 5508.153} C_VEL
LIN {X 0,Y 510.527,Z 764.288,A -85,B 0,C 180,E1 5510.66,E2 5510.66} C_VEL
LIN {X 0,Y 512.04,Z 733.931,A -85,B 0,C 180,E1 5512.525,E2 5512.525} C_VEL
LIN {X 0,Y 512.212,Z 708.406,A -85,B 0,C 180,E1 5513.602,E2 5513.602} C_VEL
LIN {X 0,Y 504.478,Z 685.03,A -85,B 0,C 180,E1 5514.682,E2 5514.682} C_VEL
LIN {X 0,Y 504.388,Z 685.03,A -85,B 0,C 180,E1 5520.569,E2 5520.569} C_VEL
LIN {X 0,Y 504.274,Z 685.03,A -85,B 0,C 180,E1 5526.76,E2 5526.76} C_VEL
LIN {X 0,Y 504.151,Z 685.03,A -85,B 0,C 180,E1 5533.505,E2 5533.505} C_VEL
LIN {X 0,Y 504.277,Z 685.03,A -85,B 0,C 180,E1 5538.837,E2 5538.837} C_VEL
LIN {X 0,Y 504.319,Z 685.03,A -85,B 0,C 180,E1 5545.362,E2 5545.362} C_VEL
LIN {X 0,Y 504.354,Z 685.03,A -85,B 0,C 180,E1 5551.406,E2 5551.406} C_VEL
LIN {X 0,Y 504.487,Z 685.03,A -85,B 0,C 180,E1 5557.123,E2 5557.123} C_VEL
LIN {X 0,Y 504.745,Z 685.03,A -85,B 0,C 180,E1 5563.075,E2 5563.075} C_VEL
LIN {X 0,Y 504.758,Z 685.03,A -85,B 0,C 180,E1 5567.925,E2 5567.925} C_VEL
LIN {X 0,Y 504.794,Z 685.03,A -85,B 0,C 180,E1 5573.137,E2 5573.137} C_VEL
LIN {X 0,Y 504.84,Z 685.03,A -85,B 0,C 180,E1 5578.291,E2 5578.291} C_VEL
LIN {X 0,Y 504.863,Z 685.03,A -85,B 0,C 180,E1 5583.431,E2 5583.431} C_VEL
LIN {X 0,Y 504.686,Z 685.03,A -85,B 0,C 180,E1 5589.355,E2 5589.355} C_VEL
LIN {X 0,Y 504.588,Z 685.03,A -85,B 0,C 180,E1 5595.616,E2 5595.616} C_VEL
LIN {X 0,Y 504.518,Z 685.03,A -85,B 0,C 180,E1 5601.036,E2 5601.036} C_VEL
LIN {X 0,Y 504.35,Z 685.03,A -85,B 0,C 180,E1 5606.668,E2 5606.668} C_VEL
LIN {X 0,Y 504.237,Z 685.03,A -85,B 0,C 180,E1 5613.077,E2 5613.077} C_VEL
LIN {X 0,Y 504.356,Z 685.03,A -85,B 0,C 180,E1 5618.931,E2 5618.931} C_VEL
LIN {X 0,Y 504.243,Z 685.03,A -85,B 0,C 180,E1 5621.826,E2 5621.826} C_VEL
LIN {X 0,Y 500.28,Z 685.03,A -85,B 0,C 180,E1 5623.774,E2 5623.774} C_VEL
LIN {X 0,Y 496.305,Z 685.03,A -85,B 0,C 180,E1 5625.753,E2 5625.753} C_VEL
LIN {X 0,Y 496.364,Z 685.177,A -85,B 0,C 180,E1 5631.126,E2 5631.126} C_VEL
LIN {X 0,Y 504.828,Z 708.453,A -85,B 0,C 180,E1 5633.21,E2 5633.21} C_VEL
LIN {X 0,Y 514.564,Z 722.331,A -85,B 0,C 180,E1 5634.696,E2 5634.696} C_VEL
LIN {X 0,Y 513.65,Z 777.212,A -85,B 0,C 180,E1 5635.677,E2 5635.677} C_VEL
LIN {X 0,Y 511.692,Z 815.094,A -85,B 0,C 180,E1 5636.999,E2 5636.999} C_VEL
LIN {X 0,Y 508.827,Z 853.526,A -85,B 0,C 180,E1 5639.064,E2 5639.064} C_VEL
LIN {X 0,Y 505.751,Z 889.255,A -85,B 0,C 180,E1 5641.784,E2 5641.784} C_VEL
LIN {X 0,Y 502.788,Z 922.029,A -85,B 0,C 180,E1 5645.156,E2 5645.156} C_VEL
LIN {X 0,Y 500.359,Z 949.792,A -85,B 0,C 180,E1 5648.949,E2 5648.949} C_VEL
LIN {X 0,Y 498.641,Z 972.477,A -85,B 0,C 180,E1 5653.068,E2 5653.068} C_VEL
LIN {X 0,Y 497.733,Z 989.57,A -85,B 0,C 180,E1 5657.305,E2 5657.305} C_VEL
LIN {X 0,Y 497.389,Z 1000.725,A -85,B 0,C 180,E1 5661.277,E2 5661.277} C_VEL
LIN {X 0,Y 497.195,Z 1006.996,A -85,B 0,C 180,E1 5664.778,E2 5664.778} C_VEL
LIN {X 0,Y 497.213,Z 1010.112,A -85,B 0,C 180,E1 5668.263,E2 5668.263} C_VEL
LIN {X 0,Y 497.298,Z 1010.11,A -85,B 0,C 180,E1 5671.742,E2 5671.742} C_VEL
LIN {X 0,Y 497.334,Z 1005.738,A -85,B 0,C 180,E1 5676.099,E2 5676.099} C_VEL
LIN {X 0,Y 497.449,Z 996.315,A -85,B 0,C 180,E1 5680.49,E2 5680.49} C_VEL
LIN {X 0,Y 498.158,Z 981.658,A -85,B 0,C 180,E1 5684.834,E2 5684.834} C_VEL
LIN {X 0,Y 499.493,Z 960.905,A -85,B 0,C 180,E1 5689.184,E2 5689.184} C_VEL
LIN {X 0,Y 501.655,Z 934.457,A -85,B 0,C 180,E1 5693.277,E2 5693.277} C_VEL
LIN {X 0,Y 504.456,Z 903.417,A -85,B 0,C 180,E1 5696.882,E2 5696.882} C_VEL
LIN {X 0,Y 507.522,Z 868.916,A -85,B 0,C 180,E1 5699.874,E2 5699.874} C_VEL
LIN {X 0,Y 510.551,Z 831.72,A -85,B 0,C 180,E1 5702.208,E2 5702.208} C_VEL
LIN {X 0,Y 512.894,Z 792.59,A -85,B 0,C 180,E1 5703.874,E2 5703.874} C_VEL
LIN {X 0,Y 514.461,Z 753.852,A -85,B 0,C 180,E1 5704.807,E2 5704.807} C_VEL
LIN {X 0,Y 514.454,Z 721.412,A -85,B 0,C 180,E1 5705.351,E2 5705.351} C_VEL
LIN {X 0,Y 501.694,Z 703.599,A -85,B 0,C 180,E1 5706.924,E2 5706.924} C_VEL
LIN {X 0,Y 496.35,Z 685.03,A -85,B 0,C 180,E1 5708.264,E2 5708.264} C_VEL
LIN {X 0,Y 496.333,Z 685.03,A -85,B 0,C 180,E1 5714.375,E2 5714.375} C_VEL
LIN {X 0,Y 496.36,Z 685.03,A -85,B 0,C 180,E1 5720.324,E2 5720.324} C_VEL
LIN {X 0,Y 496.357,Z 685.03,A -85,B 0,C 180,E1 5726.822,E2 5726.822} C_VEL
LIN {X 0,Y 496.42,Z 685.03,A -85,B 0,C 180,E1 5732.871,E2 5732.871} C_VEL
LIN {X 0,Y 496.589,Z 685.03,A -85,B 0,C 180,E1 5738.612,E2 5738.612} C_VEL
LIN {X 0,Y 496.671,Z 685.03,A -85,B 0,C 180,E1 5740.677,E2 5740.677} C_VEL
LIN {X 0,Y 503.146,Z 707.225,A -85,B 0,C 180,E1 5741.498,E2 5741.498} C_VEL
LIN {X 0,Y 502.474,Z 754.895,A -85,B 0,C 180,E1 5742.521,E2 5742.521} C_VEL
LIN {X 0,Y 501.789,Z 781.42,A -85,B 0,C 180,E1 5743.734,E2 5743.734} C_VEL
LIN {X 0,Y 500.667,Z 806.81,A -85,B 0,C 180,E1 5745.632,E2 5745.632} C_VEL
LIN {X 0,Y 499.637,Z 827.932,A -85,B 0,C 180,E1 5748.013,E2 5748.013} C_VEL
LIN {X 0,Y 498.72,Z 844.97,A -85,B 0,C 180,E1 5750.862,E2 5750.862} C_VEL
LIN {X 0,Y 498.105,Z 856.584,A -85,B 0,C 180,E1 5753.91,E2 5753.91} C_VEL
LIN {X 0,Y 497.883,Z 862.366,A -85,B 0,C 180,E1 5756.521,E2 5756.521} C_VEL
LIN {X 0,Y 497.779,Z 864.914,A -85,B 0,C 180,E1 5759.996,E2 5759.996} C_VEL
LIN {X 0,Y 497.814,Z 861.745,A -85,B 0,C 180,E1 5763.472,E2 5763.472} C_VEL
LIN {X 0,Y 498.023,Z 852.522,A -85,B 0,C 180,E1 5766.957,E2 5766.957} C_VEL
LIN {X 0,Y 498.576,Z 838.59,A -85,B 0,C 180,E1 5769.977,E2 5769.977} C_VEL
LIN {X 0,Y 499.517,Z 819.897,A -85,B 0,C 180,E1 5772.646,E2 5772.646} C_VEL
LIN {X 0,Y 500.57,Z 795.855,A -85,B 0,C 180,E1 5774.967,E2 5774.967} C_VEL
LIN {X 0,Y 501.608,Z 768.634,A -85,B 0,C 180,E1 5776.657,E2 5776.657} C_VEL
LIN {X 0,Y 502.268,Z 740.39,A -85,B 0,C 180,E1 5777.66,E2 5777.66} C_VEL
LIN {X 0,Y 501.815,Z 702.718,A -85,B 0,C 180,E1 5778.342,E2 5778.342} C_VEL
LIN {X 0,Y 496.715,Z 685.03,A -85,B 0,C 180,E1 5778.942,E2 5778.942} C_VEL
LIN {X 0,Y 496.498,Z 685.03,A -85,B 0,C 180,E1 5785.176,E2 5785.176} C_VEL
LIN {X 0,Y 496.3,Z 685.03,A -85,B 0,C 180,E1 5791.632,E2 5791.632} C_VEL
LIN {X 0,Y 496.431,Z 685.03,A -85,B 0,C 180,E1 5797.776,E2 5797.776} C_VEL
LIN {X 0,Y 496.313,Z 685.03,A -85,B 0,C 180,E1 5804.36,E2 5804.36} C_VEL
LIN {X 0,Y 496.373,Z 685.03,A -85,B 0,C 180,E1 5810.321,E2 5810.321} C_VEL
LIN {X 0,Y 496.359,Z 685.03,A -85,B 0,C 180,E1 5816.818,E2 5816.818} C_VEL
LIN {X 0,Y 496.478,Z 685.03,A -85,B 0,C 180,E1 5822.872,E2 5822.872} C_VEL
LIN {X 0,Y 496.583,Z 685.733,A -85,B 0,C 180,E1 5824.851,E2 5824.851} C_VEL
LIN {X 0,Y 505.734,Z 714.579,A -85,B 0,C 180,E1 5826.173,E2 5826.173} C_VEL
LIN {X 0,Y 504.293,Z 747.193,A -85,B 0,C 180,E1 5827.703,E2 5827.703} C_VEL
LIN {X 0,Y 502.58,Z 776.154,A -85,B 0,C 180,E1 5829.797,E2 5829.797} C_VEL
LIN {X 0,Y 500.708,Z 802.005,A -85,B 0,C 180,E1 5832.456,E2 5832.456} C_VEL
LIN {X 0,Y 499.151,Z 824.544,A -85,B 0,C 180,E1 5835.729,E2 5835.729} C_VEL
LIN {X 0,Y 498.146,Z 840.762,A -85,B 0,C 180,E1 5839.083,E2 5839.083} C_VEL
LIN {X 0,Y 497.562,Z 853.237,A -85,B 0,C 180,E1 5843.029,E2 5843.029} C_VEL
LIN {X 0,Y 497.355,Z 859.403,A -85,B 0,C 180,E1 5846.518,E2 5846.518} C_VEL
LIN {X 0,Y 497.341,Z 861.379,A -85,B 0,C 180,E1 5849.997,E2 5849.997} C_VEL
LIN {X 0,Y 497.406,Z 858.162,A -85,B 0,C 180,E1 5854.347,E2 5854.347} C_VEL
LIN {X 0,Y 497.754,Z 849.535,A -85,B 0,C 180,E1 5858.277,E2 5858.277} C_VEL
LIN {X 0,Y 498.503,Z 835.669,A -85,B 0,C 180,E1 5862.01,E2 5862.01} C_VEL
LIN {X 0,Y 499.731,Z 816.686,A -85,B 0,C 180,E1 5865.458,E2 5865.458} C_VEL
LIN {X 0,Y 501.338,Z 793.53,A -85,B 0,C 180,E1 5868.431,E2 5868.431} C_VEL
LIN {X 0,Y 503.241,Z 765.512,A -85,B 0,C 180,E1 5870.973,E2 5870.973} C_VEL
LIN {X 0,Y 504.856,Z 735.131,A -85,B 0,C 180,E1 5872.864,E2 5872.864} C_VEL
LIN {X 0,Y 505.088,Z 710.429,A -85,B 0,C 180,E1 5873.928,E2 5873.928} C_VEL
LIN {X 0,Y 496.525,Z 685.03,A -85,B 0,C 180,E1 5875.179,E2 5875.179} C_VEL
LIN {X 0,Y 496.394,Z 685.03,A -85,B 0,C 180,E1 5881.675,E2 5881.675} C_VEL
LIN {X 0,Y 496.268,Z 685.03,A -85,B 0,C 180,E1 5887.773,E2 5887.773} C_VEL
LIN {X 0,Y 496.28,Z 685.03,A -85,B 0,C 180,E1 5894.374,E2 5894.374} C_VEL
LIN {X 0,Y 496.363,Z 685.03,A -85,B 0,C 180,E1 5900.335,E2 5900.335} C_VEL
LIN {X 0,Y 496.377,Z 685.03,A -85,B 0,C 180,E1 5906.832,E2 5906.832} C_VEL
LIN {X 0,Y 496.447,Z 685.03,A -85,B 0,C 180,E1 5912.881,E2 5912.881} C_VEL
LIN {X 0,Y 496.65,Z 685.03,A -85,B 0,C 180,E1 5918.623,E2 5918.623} C_VEL
LIN {X 0,Y 496.853,Z 685.03,A -85,B 0,C 180,E1 5924.142,E2 5924.142} C_VEL
LIN {X 0,Y 496.875,Z 685.03,A -85,B 0,C 180,E1 5929.506,E2 5929.506} C_VEL
LIN {X 0,Y 496.991,Z 685.03,A -85,B 0,C 180,E1 5934.778,E2 5934.778} C_VEL
LIN {X 0,Y 497.232,Z 685.03,A -85,B 0,C 180,E1 5941.743,E2 5941.743} C_VEL
LIN {X 0,Y 496.969,Z 685.03,A -85,B 0,C 180,E1 5946.979,E2 5946.979} C_VEL
LIN {X 0,Y 496.74,Z 685.03,A -85,B 0,C 180,E1 5953.565,E2 5953.565} C_VEL
LIN {X 0,Y 496.624,Z 685.03,A -85,B 0,C 180,E1 5959.619,E2 5959.619} C_VEL
LIN {X 0,Y 496.477,Z 685.03,A -85,B 0,C 180,E1 5965.185,E2 5965.185} C_VEL
LIN {X 0,Y 496.294,Z 685.03,A -85,B 0,C 180,E1 5971.641,E2 5971.641} C_VEL
LIN {X 0,Y 496.396,Z 685.03,A -85,B 0,C 180,E1 5977.78,E2 5977.78} C_VEL
LIN {X 0,Y 496.344,Z 685.03,A -85,B 0,C 180,E1 5984.368,E2 5984.368} C_VEL
LIN {X 0,Y 496.305,Z 685.03,A -85,B 0,C 180,E1 5985.753,E2 5985.753} C_VEL
LIN {X 0,Y 492.278,Z 685.03,A -85,B 0,C 180,E1 5987.726,E2 5987.726} C_VEL
LIN {X 0,Y 488.328,Z 685.03,A -85,B 0,C 180,E1 5989.731,E2 5989.731} C_VEL
LIN {X 0,Y 488.38,Z 685.425,A -85,B 0,C 180,E1 5990.535,E2 5990.535} C_VEL
LIN {X 0,Y 498.828,Z 713.571,A -85,B 0,C 180,E1 5993.13,E2 5993.13} C_VEL
LIN {X 0,Y 506.82,Z 724.528,A -85,B 0,C 180,E1 5994.217,E2 5994.217} C_VEL
LIN {X 0,Y 507.658,Z 731.554,A -85,B 0,C 180,E1 5994.386,E2 5994.386} C_VEL
LIN {X 0,Y 506.643,Z 780.826,A -85,B 0,C 180,E1 5995.335,E2 5995.335} C_VEL
LIN {X 0,Y 504.538,Z 821.057,A -85,B 0,C 180,E1 5996.789,E2 5996.789} C_VEL
LIN {X 0,Y 501.632,Z 857.223,A -85,B 0,C 180,E1 5998.837,E2 5998.837} C_VEL
LIN {X 0,Y 498.378,Z 891.782,A -85,B 0,C 180,E1 6001.573,E2 6001.573} C_VEL
LIN {X 0,Y 495.232,Z 923.826,A -85,B 0,C 180,E1 6004.98,E2 6004.98} C_VEL
LIN {X 0,Y 492.592,Z 951.81,A -85,B 0,C 180,E1 6008.934,E2 6008.934} C_VEL
LIN {X 0,Y 490.793,Z 973.875,A -85,B 0,C 180,E1 6013.094,E2 6013.094} C_VEL
LIN {X 0,Y 489.796,Z 991.04,A -85,B 0,C 180,E1 6017.548,E2 6017.548} C_VEL
LIN {X 0,Y 489.455,Z 1002.605,A -85,B 0,C 180,E1 6022.028,E2 6022.028} C_VEL
LIN {X 0,Y 489.288,Z 1008.947,A -85,B 0,C 180,E1 6026.466,E2 6026.466} C_VEL
LIN {X 0,Y 489.311,Z 1010.5,A -85,B 0,C 180,E1 6030.003,E2 6030.003} C_VEL
LIN {X 0,Y 489.281,Z 1008.945,A -85,B 0,C 180,E1 6033.539,E2 6033.539} C_VEL
LIN {X 0,Y 489.479,Z 1002.594,A -85,B 0,C 180,E1 6037.977,E2 6037.977} C_VEL
LIN {X 0,Y 489.909,Z 991.02,A -85,B 0,C 180,E1 6042.455,E2 6042.455} C_VEL
LIN {X 0,Y 490.911,Z 973.857,A -85,B 0,C 180,E1 6046.905,E2 6046.905} C_VEL
LIN {X 0,Y 492.724,Z 950.722,A -85,B 0,C 180,E1 6051.24,E2 6051.24} C_VEL
LIN {X 0,Y 495.244,Z 923.787,A -85,B 0,C 180,E1 6055.024,E2 6055.024} C_VEL
LIN {X 0,Y 498.379,Z 891.713,A -85,B 0,C 180,E1 6058.433,E2 6058.433} C_VEL
LIN {X 0,Y 501.648,Z 857.27,A -85,B 0,C 180,E1 6061.158,E2 6061.158} C_VEL
LIN {X 0,Y 504.472,Z 821.388,A -85,B 0,C 180,E1 6063.199,E2 6063.199} C_VEL
LIN {X 0,Y 506.366,Z 782.948,A -85,B 0,C 180,E1 6064.564,E2 6064.564} C_VEL
LIN {X 0,Y 507.42,Z 736.747,A -85,B 0,C 180,E1 6065.441,E2 6065.441} C_VEL
LIN {X 0,Y 506.716,Z 724.444,A -85,B 0,C 180,E1 6065.661,E2 6065.661} C_VEL
LIN {X 0,Y 497.905,Z 712.801,A -85,B 0,C 180,E1 6066.578,E2 6066.578} C_VEL
LIN {X 0,Y 491.268,Z 696.704,A -85,B 0,C 180,E1 6067.827,E2 6067.827} C_VEL
LIN {X 0,Y 488.438,Z 685.03,A -85,B 0,C 180,E1 6068.76,E2 6068.76} C_VEL
LIN {X 0,Y 488.433,Z 685.03,A -85,B 0,C 180,E1 6075.289,E2 6075.289} C_VEL
LIN {X 0,Y 488.44,Z 685.03,A -85,B 0,C 180,E1 6081.837,E2 6081.837} C_VEL
LIN {X 0,Y 488.415,Z 685.03,A -85,B 0,C 180,E1 6088.315,E2 6088.315} C_VEL
LIN {X 0,Y 488.541,Z 685.03,A -85,B 0,C 180,E1 6094.376,E2 6094.376} C_VEL
LIN {X 0,Y 488.682,Z 685.121,A -85,B 0,C 180,E1 6100.207,E2 6100.207} C_VEL
LIN {X 0,Y 495.89,Z 708.976,A -85,B 0,C 180,E1 6101.167,E2 6101.167} C_VEL
LIN {X 0,Y 495.117,Z 757.019,A -85,B 0,C 180,E1 6102.253,E2 6102.253} C_VEL
LIN {X 0,Y 494.305,Z 784.971,A -85,B 0,C 180,E1 6103.595,E2 6103.595} C_VEL
LIN {X 0,Y 493.104,Z 809.316,A -85,B 0,C 180,E1 6105.492,E2 6105.492} C_VEL
LIN {X 0,Y 491.958,Z 831.09,A -85,B 0,C 180,E1 6108.048,E2 6108.048} C_VEL
LIN {X 0,Y 491.064,Z 846.429,A -85,B 0,C 180,E1 6110.713,E2 6110.713} C_VEL
LIN {X 0,Y 490.408,Z 858.021,A -85,B 0,C 180,E1 6113.814,E2 6113.814} C_VEL
LIN {X 0,Y 490.126,Z 863.762,A -85,B 0,C 180,E1 6116.466,E2 6116.466} C_VEL
LIN {X 0,Y 490.021,Z 866.267,A -85,B 0,C 180,E1 6119.996,E2 6119.996} C_VEL
LIN {X 0,Y 490.056,Z 863.009,A -85,B 0,C 180,E1 6123.527,E2 6123.527} C_VEL
LIN {X 0,Y 490.283,Z 853.732,A -85,B 0,C 180,E1 6127.067,E2 6127.067} C_VEL
LIN {X 0,Y 490.904,Z 839.31,A -85,B 0,C 180,E1 6130.204,E2 6130.204} C_VEL
LIN {X 0,Y 492.01,Z 819.077,A -85,B 0,C 180,E1 6133.068,E2 6133.068} C_VEL
LIN {X 0,Y 493.057,Z 795.538,A -85,B 0,C 180,E1 6135.307,E2 6135.307} C_VEL
LIN {X 0,Y 494.164,Z 768.48,A -85,B 0,C 180,E1 6136.972,E2 6136.972} C_VEL
LIN {X 0,Y 494.839,Z 739.191,A -85,B 0,C 180,E1 6137.994,E2 6137.994} C_VEL
LIN {X 0,Y 494.637,Z 705.066,A -85,B 0,C 180,E1 6138.608,E2 6138.608} C_VEL
LIN {X 0,Y 488.79,Z 685.03,A -85,B 0,C 180,E1 6139.244,E2 6139.244} C_VEL
LIN {X 0,Y 488.524,Z 685.03,A -85,B 0,C 180,E1 6145.616,E2 6145.616} C_VEL
LIN {X 0,Y 488.397,Z 685.03,A -85,B 0,C 180,E1 6151.677,E2 6151.677} C_VEL
LIN {X 0,Y 488.498,Z 685.03,A -85,B 0,C 180,E1 6158.148,E2 6158.148} C_VEL
LIN {X 0,Y 488.402,Z 685.03,A -85,B 0,C 180,E1 6164.707,E2 6164.707} C_VEL
LIN {X 0,Y 488.448,Z 685.03,A -85,B 0,C 180,E1 6170.553,E2 6170.553} C_VEL
LIN {X 0,Y 488.433,Z 685.03,A -85,B 0,C 180,E1 6176.514,E2 6176.514} C_VEL
LIN {X 0,Y 488.562,Z 685.03,A -85,B 0,C 180,E1 6182.395,E2 6182.395} C_VEL
LIN {X 0,Y 488.588,Z 685.043,A -85,B 0,C 180,E1 6184.376,E2 6184.376} C_VEL
LIN {X 0,Y 498.548,Z 716.601,A -85,B 0,C 180,E1 6185.842,E2 6185.842} C_VEL
LIN {X 0,Y 496.986,Z 749.504,A -85,B 0,C 180,E1 6187.43,E2 6187.43} C_VEL
LIN {X 0,Y 495.166,Z 778.684,A -85,B 0,C 180,E1 6189.597,E2 6189.597} C_VEL
LIN {X 0,Y 493.152,Z 805.039,A -85,B 0,C 180,E1 6192.408,E2 6192.408} C_VEL
LIN {X 0,Y 491.425,Z 827.301,A -85,B 0,C 180,E1 6195.776,E2 6195.776} C_VEL
LIN {X 0,Y 490.375,Z 843.719,A -85,B 0,C 180,E1 6199.357,E2 6199.357} C_VEL
LIN {X 0,Y 489.826,Z 854.48,A -85,B 0,C 180,E1 6202.919,E2 6202.919} C_VEL
LIN {X 0,Y 489.572,Z 860.648,A -85,B 0,C 180,E1 6206.463,E2 6206.463} C_VEL
LIN {X 0,Y 489.557,Z 862.624,A -85,B 0,C 180,E1 6209.997,E2 6209.997} C_VEL
LIN {X 0,Y 489.632,Z 859.41,A -85,B 0,C 180,E1 6214.416,E2 6214.416} C_VEL
LIN {X 0,Y 490.011,Z 850.786,A -85,B 0,C 180,E1 6218.409,E2 6218.409} C_VEL
LIN {X 0,Y 490.86,Z 836.917,A -85,B 0,C 180,E1 6222.199,E2 6222.199} C_VEL
LIN {X 0,Y 492.226,Z 817.439,A -85,B 0,C 180,E1 6225.775,E2 6225.775} C_VEL
LIN {X 0,Y 494.071,Z 793.095,A -85,B 0,C 180,E1 6228.901,E2 6228.901} C_VEL
LIN {X 0,Y 496.049,Z 765.281,A -85,B 0,C 180,E1 6231.409,E2 6231.409} C_VEL
LIN {X 0,Y 497.732,Z 735.025,A -85,B 0,C 180,E1 6233.277,E2 6233.277} C_VEL
LIN {X 0,Y 497.894,Z 712.233,A -85,B 0,C 180,E1 6234.274,E2 6234.274} C_VEL
LIN {X 0,Y 488.554,Z 685.03,A -85,B 0,C 180,E1 6235.62,E2 6235.62} C_VEL
LIN {X 0,Y 488.495,Z 685.03,A -85,B 0,C 180,E1 6241.677,E2 6241.677} C_VEL
LIN {X 0,Y 488.341,Z 685.03,A -85,B 0,C 180,E1 6248.17,E2 6248.17} C_VEL
LIN {X 0,Y 488.37,Z 685.03,A -85,B 0,C 180,E1 6254.721,E2 6254.721} C_VEL
LIN {X 0,Y 488.439,Z 685.03,A -85,B 0,C 180,E1 6260.566,E2 6260.566} C_VEL
LIN {X 0,Y 488.452,Z 685.03,A -85,B 0,C 180,E1 6266.525,E2 6266.525} C_VEL
LIN {X 0,Y 488.52,Z 685.03,A -85,B 0,C 180,E1 6272.404,E2 6272.404} C_VEL
LIN {X 0,Y 488.684,Z 685.03,A -85,B 0,C 180,E1 6278.257,E2 6278.257} C_VEL
LIN {X 0,Y 488.909,Z 685.03,A -85,B 0,C 180,E1 6283.878,E2 6283.878} C_VEL
LIN {X 0,Y 488.982,Z 685.03,A -85,B 0,C 180,E1 6289.334,E2 6289.334} C_VEL
LIN {X 0,Y 489.076,Z 685.03,A -85,B 0,C 180,E1 6294.693,E2 6294.693} C_VEL
LIN {X 0,Y 489.321,Z 685.03,A -85,B 0,C 180,E1 6301.771,E2 6301.771} C_VEL
LIN {X 0,Y 489.043,Z 685.03,A -85,B 0,C 180,E1 6307.093,E2 6307.093} C_VEL
LIN {X 0,Y 488.857,Z 685.03,A -85,B 0,C 180,E1 6312.482,E2 6312.482} C_VEL
LIN {X 0,Y 488.746,Z 685.03,A -85,B 0,C 180,E1 6317.986,E2 6317.986} C_VEL
LIN {X 0,Y 488.569,Z 685.03,A -85,B 0,C 180,E1 6323.675,E2 6323.675} C_VEL
LIN {X 0,Y 488.37,Z 685.03,A -85,B 0,C 180,E1 6330.099,E2 6330.099} C_VEL
LIN {X 0,Y 488.413,Z 685.03,A -85,B 0,C 180,E1 6335.947,E2 6335.947} C_VEL
LIN {X 0,Y 488.425,Z 685.03,A -85,B 0,C 180,E1 6342.143,E2 6342.143} C_VEL
LIN {X 0,Y 488.344,Z 685.03,A -85,B 0,C 180,E1 6347.869,E2 6347.869} C_VEL
LIN {X 0,Y 488.328,Z 685.03,A -85,B 0,C 180,E1 6349.731,E2 6349.731} C_VEL
LIN {X 0,Y 488.813,Z 688.34,A -85,B 0,C 180,E1 6350.609,E2 6350.609} C_VEL
LIN {X 0,Y 488.967,Z 699.504,A -85,B 0,C 180,E1 6351.514,E2 6351.514} C_VEL
LIN {X 0,Y 489.329,Z 711.926,A -85,B 0,C 180,E1 6352.37,E2 6352.37} C_VEL
LIN {X 0,Y 496.394,Z 724.003,A -85,B 0,C 180,E1 6353.483,E2 6353.483} C_VEL
LIN {X 0,Y 500.843,Z 729.234,A -85,B 0,C 180,E1 6353.885,E2 6353.885} C_VEL
LIN {X 0,Y 499.808,Z 778.373,A -85,B 0,C 180,E1 6354.829,E2 6354.829} C_VEL
LIN {X 0,Y 497.591,Z 818.696,A -85,B 0,C 180,E1 6356.281,E2 6356.281} C_VEL
LIN {X 0,Y 494.674,Z 857.145,A -85,B 0,C 180,E1 6358.38,E2 6358.38} C_VEL
LIN {X 0,Y 491.403,Z 890.363,A -85,B 0,C 180,E1 6360.993,E2 6360.993} C_VEL
LIN {X 0,Y 488.063,Z 922.031,A -85,B 0,C 180,E1 6364.353,E2 6364.353} C_VEL
LIN {X 0,Y 485.16,Z 950.498,A -85,B 0,C 180,E1 6368.375,E2 6368.375} C_VEL
LIN {X 0,Y 483.218,Z 972.455,A -85,B 0,C 180,E1 6372.506,E2 6372.506} C_VEL
LIN {X 0,Y 482.059,Z 989.876,A -85,B 0,C 180,E1 6376.981,E2 6376.981} C_VEL
LIN {X 0,Y 481.649,Z 1000.724,A -85,B 0,C 180,E1 6380.99,E2 6380.99} C_VEL
LIN {X 0,Y 481.415,Z 1006.997,A -85,B 0,C 180,E1 6384.607,E2 6384.607} C_VEL
LIN {X 0,Y 481.422,Z 1010.112,A -85,B 0,C 180,E1 6388.206,E2 6388.206} C_VEL
LIN {X 0,Y 481.491,Z 1010.111,A -85,B 0,C 180,E1 6391.799,E2 6391.799} C_VEL
LIN {X 0,Y 481.555,Z 1005.735,A -85,B 0,C 180,E1 6396.3,E2 6396.3} C_VEL
LIN {X 0,Y 481.723,Z 996.313,A -85,B 0,C 180,E1 6400.837,E2 6400.837} C_VEL
LIN {X 0,Y 482.62,Z 981.289,A -85,B 0,C 180,E1 6405.416,E2 6405.416} C_VEL
LIN {X 0,Y 484.17,Z 960.902,A -85,B 0,C 180,E1 6409.816,E2 6409.816} C_VEL
LIN {X 0,Y 486.562,Z 936.274,A -85,B 0,C 180,E1 6413.781,E2 6413.781} C_VEL
LIN {X 0,Y 489.806,Z 905.435,A -85,B 0,C 180,E1 6417.529,E2 6417.529} C_VEL
LIN {X 0,Y 493.258,Z 872.22,A -85,B 0,C 180,E1 6420.548,E2 6420.548} C_VEL
LIN {X 0,Y 495.907,Z 839.944,A -85,B 0,C 180,E1 6422.632,E2 6422.632} C_VEL
LIN {X 0,Y 498.307,Z 799.169,A -85,B 0,C 180,E1 6424.405,E2 6424.405} C_VEL
LIN {X 0,Y 500.062,Z 756.891,A -85,B 0,C 180,E1 6425.496,E2 6425.496} C_VEL
LIN {X 0,Y 499.465,Z 727.963,A -85,B 0,C 180,E1 6425.99,E2 6425.99} C_VEL
LIN {X 0,Y 490.062,Z 715.158,A -85,B 0,C 180,E1 6426.813,E2 6426.813} C_VEL
LIN {X 0,Y 483.132,Z 695.502,A -85,B 0,C 180,E1 6428.332,E2 6428.332} C_VEL
LIN {X 0,Y 480.473,Z 685.03,A -85,B 0,C 180,E1 6429.219,E2 6429.219} C_VEL
LIN {X 0,Y 480.488,Z 685.03,A -85,B 0,C 180,E1 6436.296,E2 6436.296} C_VEL
LIN {X 0,Y 480.559,Z 685.03,A -85,B 0,C 180,E1 6441.731,E2 6441.731} C_VEL
LIN {X 0,Y 480.502,Z 685.03,A -85,B 0,C 180,E1 6447.997,E2 6447.997} C_VEL
LIN {X 0,Y 480.629,Z 685.03,A -85,B 0,C 180,E1 6453.923,E2 6453.923} C_VEL
LIN {X 0,Y 480.737,Z 685.03,A -85,B 0,C 180,E1 6459.679,E2 6459.679} C_VEL
LIN {X 0,Y 488.717,Z 709.736,A -85,B 0,C 180,E1 6460.798,E2 6460.798} C_VEL
LIN {X 0,Y 487.742,Z 759.287,A -85,B 0,C 180,E1 6461.975,E2 6461.975} C_VEL
LIN {X 0,Y 486.923,Z 786.833,A -85,B 0,C 180,E1 6463.339,E2 6463.339} C_VEL
LIN {X 0,Y 485.59,Z 811.592,A -85,B 0,C 180,E1 6465.325,E2 6465.325} C_VEL
LIN {X 0,Y 484.389,Z 832.642,A -85,B 0,C 180,E1 6467.858,E2 6467.858} C_VEL
LIN {X 0,Y 483.392,Z 848.346,A -85,B 0,C 180,E1 6470.657,E2 6470.657} C_VEL
LIN {X 0,Y 482.709,Z 859.463,A -85,B 0,C 180,E1 6473.715,E2 6473.715} C_VEL
LIN {X 0,Y 482.396,Z 865.161,A -85,B 0,C 180,E1 6476.409,E2 6476.409} C_VEL
LIN {X 0,Y 482.266,Z 867.608,A -85,B 0,C 180,E1 6479.996,E2 6479.996} C_VEL
LIN {X 0,Y 482.273,Z 864.283,A -85,B 0,C 180,E1 6483.584,E2 6483.584} C_VEL
LIN {X 0,Y 482.557,Z 854.925,A -85,B 0,C 180,E1 6487.181,E2 6487.181} C_VEL
LIN {X 0,Y 483.234,Z 840.431,A -85,B 0,C 180,E1 6490.368,E2 6490.368} C_VEL
LIN {X 0,Y 484.388,Z 820.136,A -85,B 0,C 180,E1 6493.277,E2 6493.277} C_VEL
LIN {X 0,Y 485.548,Z 796.271,A -85,B 0,C 180,E1 6495.571,E2 6495.571} C_VEL
LIN {X 0,Y 486.711,Z 768.325,A -85,B 0,C 180,E1 6497.299,E2 6497.299} C_VEL
LIN {X 0,Y 487.415,Z 738.758,A -85,B 0,C 180,E1 6498.316,E2 6498.316} C_VEL
LIN {X 0,Y 486.885,Z 705.377,A -85,B 0,C 180,E1 6498.944,E2 6498.944} C_VEL
LIN {X 0,Y 480.868,Z 685.03,A -85,B 0,C 180,E1 6499.692,E2 6499.692} C_VEL
LIN {X 0,Y 480.609,Z 685.03,A -85,B 0,C 180,E1 6506.069,E2 6506.069} C_VEL
LIN {X 0,Y 480.483,Z 685.03,A -85,B 0,C 180,E1 6512.262,E2 6512.262} C_VEL
LIN {X 0,Y 480.564,Z 685.03,A -85,B 0,C 180,E1 6518.894,E2 6518.894} C_VEL
LIN {X 0,Y 480.441,Z 685.03,A -85,B 0,C 180,E1 6523.74,E2 6523.74} C_VEL
LIN {X 0,Y 480.475,Z 685.03,A -85,B 0,C 180,E1 6528.905,E2 6528.905} C_VEL
LIN {X 0,Y 480.474,Z 685.03,A -85,B 0,C 180,E1 6534.729,E2 6534.729} C_VEL
LIN {X 0,Y 480.556,Z 685.03,A -85,B 0,C 180,E1 6539.835,E2 6539.835} C_VEL
LIN {X 0,Y 480.66,Z 685.03,A -85,B 0,C 180,E1 6543.877,E2 6543.877} C_VEL
LIN {X 0,Y 491.407,Z 717.743,A -85,B 0,C 180,E1 6545.469,E2 6545.469} C_VEL
LIN {X 0,Y 489.915,Z 749.458,A -85,B 0,C 180,E1 6547.005,E2 6547.005} C_VEL
LIN {X 0,Y 487.954,Z 778.575,A -85,B 0,C 180,E1 6549.163,E2 6549.163} C_VEL
LIN {X 0,Y 485.824,Z 804.46,A -85,B 0,C 180,E1 6551.9,E2 6551.9} C_VEL
LIN {X 0,Y 484.183,Z 825.582,A -85,B 0,C 180,E1 6555.014,E2 6555.014} C_VEL
LIN {X 0,Y 482.825,Z 843.245,A -85,B 0,C 180,E1 6558.732,E2 6558.732} C_VEL
LIN {X 0,Y 482.092,Z 855.724,A -85,B 0,C 180,E1 6562.804,E2 6562.804} C_VEL
LIN {X 0,Y 481.808,Z 861.891,A -85,B 0,C 180,E1 6566.406,E2 6566.406} C_VEL
LIN {X 0,Y 481.774,Z 863.869,A -85,B 0,C 180,E1 6569.997,E2 6569.997} C_VEL
LIN {X 0,Y 481.871,Z 860.655,A -85,B 0,C 180,E1 6574.488,E2 6574.488} C_VEL
LIN {X 0,Y 482.302,Z 852.032,A -85,B 0,C 180,E1 6578.544,E2 6578.544} C_VEL
LIN {X 0,Y 483.21,Z 838.166,A -85,B 0,C 180,E1 6582.396,E2 6582.396} C_VEL
LIN {X 0,Y 484.654,Z 819.683,A -85,B 0,C 180,E1 6585.873,E2 6585.873} C_VEL
LIN {X 0,Y 486.586,Z 795.616,A -85,B 0,C 180,E1 6589.056,E2 6589.056} C_VEL
LIN {X 0,Y 488.714,Z 767.952,A -85,B 0,C 180,E1 6591.627,E2 6591.627} C_VEL
LIN {X 0,Y 490.504,Z 737.529,A -85,B 0,C 180,E1 6593.573,E2 6593.573} C_VEL
LIN {X 0,Y 490.805,Z 714.263,A -85,B 0,C 180,E1 6594.615,E2 6594.615} C_VEL
LIN {X 0,Y 480.634,Z 685.03,A -85,B 0,C 180,E1 6596.073,E2 6596.073} C_VEL
LIN {X 0,Y 480.566,Z 685.03,A -85,B 0,C 180,E1 6602.262,E2 6602.262} C_VEL
LIN {X 0,Y 480.424,Z 685.03,A -85,B 0,C 180,E1 6608.916,E2 6608.916} C_VEL
LIN {X 0,Y 480.405,Z 685.03,A -85,B 0,C 180,E1 6613.754,E2 6613.754} C_VEL
LIN {X 0,Y 480.465,Z 685.03,A -85,B 0,C 180,E1 6618.917,E2 6618.917} C_VEL
LIN {X 0,Y 480.487,Z 685.03,A -85,B 0,C 180,E1 6624.74,E2 6624.74} C_VEL
LIN {X 0,Y 480.525,Z 685.03,A -85,B 0,C 180,E1 6629.845,E2 6629.845} C_VEL
LIN {X 0,Y 480.661,Z 685.03,A -85,B 0,C 180,E1 6635.919,E2 6635.919} C_VEL
LIN {X 0,Y 480.886,Z 685.03,A -85,B 0,C 180,E1 6641.718,E2 6641.718} C_VEL
LIN {X 0,Y 481.048,Z 685.03,A -85,B 0,C 180,E1 6647.321,E2 6647.321} C_VEL
LIN {X 0,Y 481.082,Z 685.03,A -85,B 0,C 180,E1 6652.797,E2 6652.797} C_VEL
LIN {X 0,Y 481.184,Z 685.03,A -85,B 0,C 180,E1 6658.207,E2 6658.207} C_VEL
LIN {X 0,Y 481.195,Z 685.03,A -85,B 0,C 180,E1 6663.6,E2 6663.6} C_VEL
LIN {X 0,Y 480.995,Z 685.03,A -85,B 0,C 180,E1 6669.028,E2 6669.028} C_VEL
LIN {X 0,Y 480.882,Z 685.03,A -85,B 0,C 180,E1 6674.542,E2 6674.542} C_VEL
LIN {X 0,Y 480.763,Z 685.03,A -85,B 0,C 180,E1 6680.2,E2 6680.2} C_VEL
LIN {X 0,Y 480.593,Z 685.03,A -85,B 0,C 180,E1 6686.079,E2 6686.079} C_VEL
LIN {X 0,Y 480.483,Z 685.03,A -85,B 0,C 180,E1 6692.271,E2 6692.271} C_VEL
LIN {X 0,Y 480.554,Z 685.03,A -85,B 0,C 180,E1 6698.906,E2 6698.906} C_VEL
LIN {X 0,Y 480.455,Z 685.03,A -85,B 0,C 180,E1 6703.75,E2 6703.75} C_VEL
LIN {X 0,Y 480.464,Z 685.802,A -85,B 0,C 180,E1 6709.935,E2 6709.935} C_VEL
LIN {X 0,Y 489.329,Z 711.926,A -85,B 0,C 180,E1 6712.37,E2 6712.37} C_VEL
LIN {X 0,Y 492.716,Z 725.235,A -85,B 0,C 180,E1 6713.179,E2 6713.179} C_VEL
LIN {X 0,Y 493.98,Z 744.876,A -85,B 0,C 180,E1 6713.663,E2 6713.663} C_VEL
LIN {X 0,Y 492.513,Z 785.84,A -85,B 0,C 180,E1 6714.603,E2 6714.603} C_VEL
LIN {X 0,Y 489.972,Z 825.982,A -85,B 0,C 180,E1 6716.216,E2 6716.216} C_VEL
LIN {X 0,Y 486.827,Z 863.729,A -85,B 0,C 180,E1 6718.462,E2 6718.462} C_VEL
LIN {X 0,Y 483.601,Z 897.501,A -85,B 0,C 180,E1 6721.222,E2 6721.222} C_VEL
LIN {X 0,Y 480.085,Z 927.629,A -85,B 0,C 180,E1 6724.644,E2 6724.644} C_VEL
LIN {X 0,Y 477.135,Z 954.607,A -85,B 0,C 180,E1 6728.713,E2 6728.713} C_VEL
LIN {X 0,Y 475.112,Z 976.274,A -85,B 0,C 180,E1 6733.086,E2 6733.086} C_VEL
LIN {X 0,Y 474.048,Z 992.435,A -85,B 0,C 180,E1 6737.594,E2 6737.594} C_VEL
LIN {X 0,Y 473.68,Z 1002.633,A -85,B 0,C 180,E1 6741.775,E2 6741.775} C_VEL
LIN {X 0,Y 473.483,Z 1008.945,A -85,B 0,C 180,E1 6746.348,E2 6746.348} C_VEL
LIN {X 0,Y 473.522,Z 1010.5,A -85,B 0,C 180,E1 6750.003,E2 6750.003} C_VEL
LIN {X 0,Y 473.485,Z 1008.941,A -85,B 0,C 180,E1 6753.658,E2 6753.658} C_VEL
LIN {X 0,Y 473.705,Z 1002.62,A -85,B 0,C 180,E1 6758.231,E2 6758.231} C_VEL
LIN {X 0,Y 474.315,Z 990.005,A -85,B 0,C 180,E1 6763.195,E2 6763.195} C_VEL
LIN {X 0,Y 475.523,Z 972.287,A -85,B 0,C 180,E1 6767.825,E2 6767.825} C_VEL
LIN {X 0,Y 477.79,Z 948.748,A -85,B 0,C 180,E1 6772.276,E2 6772.276} C_VEL
LIN {X 0,Y 480.876,Z 920.734,A -85,B 0,C 180,E1 6776.23,E2 6776.23} C_VEL
LIN {X 0,Y 484.283,Z 890.491,A -85,B 0,C 180,E1 6779.433,E2 6779.433} C_VEL
LIN {X 0,Y 487.16,Z 857.242,A -85,B 0,C 180,E1 6781.906,E2 6781.906} C_VEL
LIN {X 0,Y 489.9,Z 817.698,A -85,B 0,C 180,E1 6784.009,E2 6784.009} C_VEL
LIN {X 0,Y 492.132,Z 776.417,A -85,B 0,C 180,E1 6785.436,E2 6785.436} C_VEL
LIN {X 0,Y 492.508,Z 731.611,A -85,B 0,C 180,E1 6786.311,E2 6786.311} C_VEL
LIN {X 0,Y 480.714,Z 713.877,A -85,B 0,C 180,E1 6787.356,E2 6787.356} C_VEL
LIN {X 0,Y 472.529,Z 685.03,A -85,B 0,C 180,E1 6789.7,E2 6789.7} C_VEL
LIN {X 0,Y 472.485,Z 685.03,A -85,B 0,C 180,E1 6795.361,E2 6795.361} C_VEL
LIN {X 0,Y 472.543,Z 685.03,A -85,B 0,C 180,E1 6800.306,E2 6800.306} C_VEL
LIN {X 0,Y 472.534,Z 685.03,A -85,B 0,C 180,E1 6806.138,E2 6806.138} C_VEL
LIN {X 0,Y 472.589,Z 685.03,A -85,B 0,C 180,E1 6811.381,E2 6811.381} C_VEL
LIN {X 0,Y 472.789,Z 685.03,A -85,B 0,C 180,E1 6817.773,E2 6817.773} C_VEL
LIN {X 0,Y 472.834,Z 685.073,A -85,B 0,C 180,E1 6819.134,E2 6819.134} C_VEL
LIN {X 0,Y 481.592,Z 710.885,A -85,B 0,C 180,E1 6820.417,E2 6820.417} C_VEL
LIN {X 0,Y 480.417,Z 761.752,A -85,B 0,C 180,E1 6821.691,E2 6821.691} C_VEL
LIN {X 0,Y 479.548,Z 788.742,A -85,B 0,C 180,E1 6823.075,E2 6823.075} C_VEL
LIN {X 0,Y 478.132,Z 813.305,A -85,B 0,C 180,E1 6825.09,E2 6825.09} C_VEL
LIN {X 0,Y 476.827,Z 834.222,A -85,B 0,C 180,E1 6827.663,E2 6827.663} C_VEL
LIN {X 0,Y 475.706,Z 850.202,A -85,B 0,C 180,E1 6830.586,E2 6830.586} C_VEL
LIN {X 0,Y 474.887,Z 862.111,A -85,B 0,C 180,E1 6834.069,E2 6834.069} C_VEL
LIN {X 0,Y 474.638,Z 866.57,A -85,B 0,C 180,E1 6836.351,E2 6836.351} C_VEL
LIN {X 0,Y 474.508,Z 868.951,A -85,B 0,C 180,E1 6839.996,E2 6839.996} C_VEL
LIN {X 0,Y 474.515,Z 865.558,A -85,B 0,C 180,E1 6843.642,E2 6843.642} C_VEL
LIN {X 0,Y 474.815,Z 856.121,A -85,B 0,C 180,E1 6847.299,E2 6847.299} C_VEL
LIN {X 0,Y 475.581,Z 841.133,A -85,B 0,C 180,E1 6850.61,E2 6850.61} C_VEL
LIN {X 0,Y 476.788,Z 821.183,A -85,B 0,C 180,E1 6853.493,E2 6853.493} C_VEL
LIN {X 0,Y 478.021,Z 796.968,A -85,B 0,C 180,E1 6855.845,E2 6855.845} C_VEL
LIN {X 0,Y 479.24,Z 769.292,A -85,B 0,C 180,E1 6857.577,E2 6857.577} C_VEL
LIN {X 0,Y 479.945,Z 740.927,A -85,B 0,C 180,E1 6858.587,E2 6858.587} C_VEL
LIN {X 0,Y 479.541,Z 707.054,A -85,B 0,C 180,E1 6859.244,E2 6859.244} C_VEL
LIN {X 0,Y 472.904,Z 685.03,A -85,B 0,C 180,E1 6860.078,E2 6860.078} C_VEL
LIN {X 0,Y 472.637,Z 685.03,A -85,B 0,C 180,E1 6866.612,E2 6866.612} C_VEL
LIN {X 0,Y 472.51,Z 685.03,A -85,B 0,C 180,E1 6872.874,E2 6872.874} C_VEL
LIN {X 0,Y 472.651,Z 685.03,A -85,B 0,C 180,E1 6877.335,E2 6877.335} C_VEL
LIN {X 0,Y 472.463,Z 685.03,A -85,B 0,C 180,E1 6882.719,E2 6882.719} C_VEL
LIN {X 0,Y 472.482,Z 685.03,A -85,B 0,C 180,E1 6887.873,E2 6887.873} C_VEL
LIN {X 0,Y 472.617,Z 685.03,A -85,B 0,C 180,E1 6892.947,E2 6892.947} C_VEL
LIN {X 0,Y 472.637,Z 685.03,A -85,B 0,C 180,E1 6899.53,E2 6899.53} C_VEL
LIN {X 0,Y 472.766,Z 685.03,A -85,B 0,C 180,E1 6903.408,E2 6903.408} C_VEL
LIN {X 0,Y 484.076,Z 718.876,A -85,B 0,C 180,E1 6905.069,E2 6905.069} C_VEL
LIN {X 0,Y 482.667,Z 751.478,A -85,B 0,C 180,E1 6906.694,E2 6906.694} C_VEL
LIN {X 0,Y 480.569,Z 781.105,A -85,B 0,C 180,E1 6908.948,E2 6908.948} C_VEL
LIN {X 0,Y 478.295,Z 807.489,A -85,B 0,C 180,E1 6911.843,E2 6911.843} C_VEL
LIN {X 0,Y 476.476,Z 828.298,A -85,B 0,C 180,E1 6915.043,E2 6915.043} C_VEL
LIN {X 0,Y 475.186,Z 844.483,A -85,B 0,C 180,E1 6918.549,E2 6918.549} C_VEL
LIN {X 0,Y 474.356,Z 856.967,A -85,B 0,C 180,E1 6922.686,E2 6922.686} C_VEL
LIN {X 0,Y 474.026,Z 863.137,A -85,B 0,C 180,E1 6926.347,E2 6926.347} C_VEL
LIN {X 0,Y 473.991,Z 865.114,A -85,B 0,C 180,E1 6929.997,E2 6929.997} C_VEL
LIN {X 0,Y 474.116,Z 861.899,A -85,B 0,C 180,E1 6934.561,E2 6934.561} C_VEL
LIN {X 0,Y 474.563,Z 853.283,A -85,B 0,C 180,E1 6938.685,E2 6938.685} C_VEL
LIN {X 0,Y 475.557,Z 839.416,A -85,B 0,C 180,E1 6942.598,E2 6942.598} C_VEL
LIN {X 0,Y 477.185,Z 820.422,A -85,B 0,C 180,E1 6946.207,E2 6946.207} C_VEL
LIN {X 0,Y 479.175,Z 797.271,A -85,B 0,C 180,E1 6949.311,E2 6949.311} C_VEL
LIN {X 0,Y 481.478,Z 769.175,A -85,B 0,C 180,E1 6951.969,E2 6951.969} C_VEL
LIN {X 0,Y 483.377,Z 738.735,A -85,B 0,C 180,E1 6953.942,E2 6953.942} C_VEL
LIN {X 0,Y 483.748,Z 716.705,A -85,B 0,C 180,E1 6954.948,E2 6954.948} C_VEL
LIN {X 0,Y 472.662,Z 685.03,A -85,B 0,C 180,E1 6956.547,E2 6956.547} C_VEL
LIN {X 0,Y 472.572,Z 685.03,A -85,B 0,C 180,E1 6962.876,E2 6962.876} C_VEL
LIN {X 0,Y 472.55,Z 685.03,A -85,B 0,C 180,E1 6967.352,E2 6967.352} C_VEL
LIN {X 0,Y 472.434,Z 685.03,A -85,B 0,C 180,E1 6974.643,E2 6974.643} C_VEL
LIN {X 0,Y 472.534,Z 685.03,A -85,B 0,C 180,E1 6980.316,E2 6980.316} C_VEL
LIN {X 0,Y 472.534,Z 685.03,A -85,B 0,C 180,E1 6986.128,E2 6986.128} C_VEL
LIN {X 0,Y 472.637,Z 685.03,A -85,B 0,C 180,E1 6991.393,E2 6991.393} C_VEL
LIN {X 0,Y 472.847,Z 685.03,A -85,B 0,C 180,E1 6997.741,E2 6997.741} C_VEL
LIN {X 0,Y 473.034,Z 685.03,A -85,B 0,C 180,E1 7003.321,E2 7003.321} C_VEL
LIN {X 0,Y 473.153,Z 685.03,A -85,B 0,C 180,E1 7008.973,E2 7008.973} C_VEL
LIN {X 0,Y 473.245,Z 685.03,A -85,B 0,C 180,E1 7014.515,E2 7014.515} C_VEL
LIN {X 0,Y 473.445,Z 685.03,A -85,B 0,C 180,E1 7020.004,E2 7020.004} C_VEL
LIN {X 0,Y 473.256,Z 685.03,A -85,B 0,C 180,E1 7025.493,E2 7025.493} C_VEL
LIN {X 0,Y 473.034,Z 685.03,A -85,B 0,C 180,E1 7031.038,E2 7031.038} C_VEL
LIN {X 0,Y 472.9,Z 685.03,A -85,B 0,C 180,E1 7036.807,E2 7036.807} C_VEL
LIN {X 0,Y 472.783,Z 685.03,A -85,B 0,C 180,E1 7042.523,E2 7042.523} C_VEL
LIN {X 0,Y 472.56,Z 685.03,A -85,B 0,C 180,E1 7048.621,E2 7048.621} C_VEL
LIN {X 0,Y 472.584,Z 685.03,A -85,B 0,C 180,E1 7055.084,E2 7055.084} C_VEL
LIN {X 0,Y 472.547,Z 685.03,A -85,B 0,C 180,E1 7059.969,E2 7059.969} C_VEL
LIN {X 0,Y 472.455,Z 685.03,A -85,B 0,C 180,E1 7065.359,E2 7065.359} C_VEL
LIN {X 0,Y 472.532,Z 685.307,A -85,B 0,C 180,E1 7069.26,E2 7069.26} C_VEL
LIN {X 0,Y 485.512,Z 721.327,A -85,B 0,C 180,E1 7072.63,E2 7072.63} C_VEL
LIN {X 0,Y 494.026,Z 732.871,A -85,B 0,C 180,E1 7073.467,E2 7073.467} C_VEL
LIN {X 0,Y 493.98,Z 744.876,A -85,B 0,C 180,E1 7073.663,E2 7073.663} C_VEL
LIN {X 0,Y 490.117,Z 762.014,A -85,B 0,C 180,E1 7073.734,E2 7073.734} C_VEL
LIN {X 0,Y 486.212,Z 776.846,A -85,B 0,C 180,E1 7073.877,E2 7073.877} C_VEL
LIN {X 0,Y 486.042,Z 778.925,A -85,B 0,C 180,E1 7073.936,E2 7073.936} C_VEL
LIN {X 0,Y 483.48,Z 818.245,A -85,B 0,C 180,E1 7075.414,E2 7075.414} C_VEL
LIN {X 0,Y 479.984,Z 858.153,A -85,B 0,C 180,E1 7077.694,E2 7077.694} C_VEL
LIN {X 0,Y 476.329,Z 895.085,A -85,B 0,C 180,E1 7080.657,E2 7080.657} C_VEL
LIN {X 0,Y 473.208,Z 923.906,A -85,B 0,C 180,E1 7083.741,E2 7083.741} C_VEL
LIN {X 0,Y 469.99,Z 951.209,A -85,B 0,C 180,E1 7087.765,E2 7087.765} C_VEL
LIN {X 0,Y 467.617,Z 974.199,A -85,B 0,C 180,E1 7092.304,E2 7092.304} C_VEL
LIN {X 0,Y 466.327,Z 991.038,A -85,B 0,C 180,E1 7096.91,E2 7096.91} C_VEL
LIN {X 0,Y 465.815,Z 1002.866,A -85,B 0,C 180,E1 7101.757,E2 7101.757} C_VEL
LIN {X 0,Y 465.604,Z 1008.944,A -85,B 0,C 180,E1 7106.286,E2 7106.286} C_VEL
LIN {X 0,Y 465.634,Z 1010.5,A -85,B 0,C 180,E1 7110.003,E2 7110.003} C_VEL
LIN {X 0,Y 465.609,Z 1008.937,A -85,B 0,C 180,E1 7113.719,E2 7113.719} C_VEL
LIN {X 0,Y 465.839,Z 1002.839,A -85,B 0,C 180,E1 7118.255,E2 7118.255} C_VEL
LIN {X 0,Y 466.409,Z 991.017,A -85,B 0,C 180,E1 7123.093,E2 7123.093} C_VEL
LIN {X 0,Y 467.734,Z 972.967,A -85,B 0,C 180,E1 7127.975,E2 7127.975} C_VEL
LIN {X 0,Y 470.128,Z 949.953,A -85,B 0,C 180,E1 7132.448,E2 7132.448} C_VEL
LIN {X 0,Y 473.42,Z 921.942,A -85,B 0,C 180,E1 7136.507,E2 7136.507} C_VEL
LIN {X 0,Y 476.278,Z 894.324,A -85,B 0,C 180,E1 7139.355,E2 7139.355} C_VEL
LIN {X 0,Y 479.577,Z 857.754,A -85,B 0,C 180,E1 7142.149,E2 7142.149} C_VEL
LIN {X 0,Y 482.498,Z 817.87,A -85,B 0,C 180,E1 7144.329,E2 7144.329} C_VEL
LIN {X 0,Y 484.883,Z 776.604,A -85,B 0,C 180,E1 7145.798,E2 7145.798} C_VEL
LIN {X 0,Y 485.178,Z 734.653,A -85,B 0,C 180,E1 7146.673,E2 7146.673} C_VEL
LIN {X 0,Y 472.903,Z 714.966,A -85,B 0,C 180,E1 7147.772,E2 7147.772} C_VEL
LIN {X 0,Y 464.598,Z 685.03,A -85,B 0,C 180,E1 7150.194,E2 7150.194} C_VEL
LIN {X 0,Y 464.601,Z 685.03,A -85,B 0,C 180,E1 7156.993,E2 7156.993} C_VEL
LIN {X 0,Y 464.614,Z 685.03,A -85,B 0,C 180,E1 7161.894,E2 7161.894} C_VEL
LIN {X 0,Y 464.572,Z 685.03,A -85,B 0,C 180,E1 7168.686,E2 7168.686} C_VEL
LIN {X 0,Y 464.826,Z 685.03,A -85,B 0,C 180,E1 7175.379,E2 7175.379} C_VEL
LIN {X 0,Y 464.93,Z 685.336,A -85,B 0,C 180,E1 7178.532,E2 7178.532} C_VEL
LIN {X 0,Y 474.448,Z 713.002,A -85,B 0,C 180,E1 7180.036,E2 7180.036} C_VEL
LIN {X 0,Y 473.182,Z 763.167,A -85,B 0,C 180,E1 7181.357,E2 7181.357} C_VEL
LIN {X 0,Y 472.204,Z 790.776,A -85,B 0,C 180,E1 7182.804,E2 7182.804} C_VEL
LIN {X 0,Y 470.696,Z 815.533,A -85,B 0,C 180,E1 7184.899,E2 7184.899} C_VEL
LIN {X 0,Y 469.291,Z 835.843,A -85,B 0,C 180,E1 7187.461,E2 7187.461} C_VEL
LIN {X 0,Y 468.064,Z 851.743,A -85,B 0,C 180,E1 7190.431,E2 7190.431} C_VEL
LIN {X 0,Y 467.182,Z 863.559,A -85,B 0,C 180,E1 7193.971,E2 7193.971} C_VEL
LIN {X 0,Y 466.909,Z 867.981,A -85,B 0,C 180,E1 7196.29,E2 7196.29} C_VEL
LIN {X 0,Y 466.726,Z 870.301,A -85,B 0,C 180,E1 7199.996,E2 7199.996} C_VEL
LIN {X 0,Y 466.738,Z 866.824,A -85,B 0,C 180,E1 7203.703,E2 7203.703} C_VEL
LIN {X 0,Y 467.089,Z 857.302,A -85,B 0,C 180,E1 7207.42,E2 7207.42} C_VEL
LIN {X 0,Y 467.9,Z 842.223,A -85,B 0,C 180,E1 7210.786,E2 7210.786} C_VEL
LIN {X 0,Y 469.163,Z 822.204,A -85,B 0,C 180,E1 7213.716,E2 7213.716} C_VEL
LIN {X 0,Y 470.463,Z 798.382,A -85,B 0,C 180,E1 7216.069,E2 7216.069} C_VEL
LIN {X 0,Y 471.783,Z 770.215,A -85,B 0,C 180,E1 7217.864,E2 7217.864} C_VEL
LIN {X 0,Y 472.523,Z 742.245,A -85,B 0,C 180,E1 7218.881,E2 7218.881} C_VEL
LIN {X 0,Y 472.292,Z 709.079,A -85,B 0,C 180,E1 7219.542,E2 7219.542} C_VEL
LIN {X 0,Y 464.97,Z 685.03,A -85,B 0,C 180,E1 7220.475,E2 7220.475} C_VEL
LIN {X 0,Y 464.695,Z 685.03,A -85,B 0,C 180,E1 7227.033,E2 7227.033} C_VEL
LIN {X 0,Y 464.605,Z 685.03,A -85,B 0,C 180,E1 7233.506,E2 7233.506} C_VEL
LIN {X 0,Y 464.602,Z 685.03,A -85,B 0,C 180,E1 7238.776,E2 7238.776} C_VEL
LIN {X 0,Y 464.548,Z 685.03,A -85,B 0,C 180,E1 7245.602,E2 7245.602} C_VEL
LIN {X 0,Y 464.61,Z 685.03,A -85,B 0,C 180,E1 7251.89,E2 7251.89} C_VEL
LIN {X 0,Y 464.619,Z 685.03,A -85,B 0,C 180,E1 7258.686,E2 7258.686} C_VEL
LIN {X 0,Y 464.807,Z 685.377,A -85,B 0,C 180,E1 7262.905,E2 7262.905} C_VEL
LIN {X 0,Y 476.408,Z 718.737,A -85,B 0,C 180,E1 7264.582,E2 7264.582} C_VEL
LIN {X 0,Y 476.334,Z 738.963,A -85,B 0,C 180,E1 7265.537,E2 7265.537} C_VEL
LIN {X 0,Y 474.262,Z 769.96,A -85,B 0,C 180,E1 7267.55,E2 7267.55} C_VEL
LIN {X 0,Y 471.956,Z 797.56,A -85,B 0,C 180,E1 7270.175,E2 7270.175} C_VEL
LIN {X 0,Y 469.711,Z 821.613,A -85,B 0,C 180,E1 7273.43,E2 7273.43} C_VEL
LIN {X 0,Y 467.922,Z 841.022,A -85,B 0,C 180,E1 7277.187,E2 7277.187} C_VEL
LIN {X 0,Y 466.829,Z 854.752,A -85,B 0,C 180,E1 7281.164,E2 7281.164} C_VEL
LIN {X 0,Y 466.346,Z 863.26,A -85,B 0,C 180,E1 7285.357,E2 7285.357} C_VEL
LIN {X 0,Y 466.19,Z 866.361,A -85,B 0,C 180,E1 7289.997,E2 7289.997} C_VEL
LIN {X 0,Y 466.348,Z 863.146,A -85,B 0,C 180,E1 7294.637,E2 7294.637} C_VEL
LIN {X 0,Y 466.847,Z 854.53,A -85,B 0,C 180,E1 7298.829,E2 7298.829} C_VEL
LIN {X 0,Y 467.938,Z 840.661,A -85,B 0,C 180,E1 7302.807,E2 7302.807} C_VEL
LIN {X 0,Y 469.601,Z 822.583,A -85,B 0,C 180,E1 7306.328,E2 7306.328} C_VEL
LIN {X 0,Y 471.767,Z 799.087,A -85,B 0,C 180,E1 7309.556,E2 7309.556} C_VEL
LIN {X 0,Y 474.134,Z 771.862,A -85,B 0,C 180,E1 7312.204,E2 7312.204} C_VEL
LIN {X 0,Y 476.224,Z 741.051,A -85,B 0,C 180,E1 7314.264,E2 7314.264} C_VEL
LIN {X 0,Y 476.571,Z 718.646,A -85,B 0,C 180,E1 7315.32,E2 7315.32} C_VEL
LIN {X 0,Y 464.746,Z 685.03,A -85,B 0,C 180,E1 7317.036,E2 7317.036} C_VEL
LIN {X 0,Y 464.645,Z 685.03,A -85,B 0,C 180,E1 7323.51,E2 7323.51} C_VEL
LIN {X 0,Y 464.497,Z 685.03,A -85,B 0,C 180,E1 7328.781,E2 7328.781} C_VEL
LIN {X 0,Y 464.518,Z 685.03,A -85,B 0,C 180,E1 7335.616,E2 7335.616} C_VEL
LIN {X 0,Y 464.607,Z 685.03,A -85,B 0,C 180,E1 7341.904,E2 7341.904} C_VEL
LIN {X 0,Y 464.61,Z 685.03,A -85,B 0,C 180,E1 7348.698,E2 7348.698} C_VEL
LIN {X 0,Y 464.831,Z 685.03,A -85,B 0,C 180,E1 7355.364,E2 7355.364} C_VEL
LIN {X 0,Y 465.004,Z 685.03,A -85,B 0,C 180,E1 7361.07,E2 7361.07} C_VEL
LIN {X 0,Y 465.221,Z 685.03,A -85,B 0,C 180,E1 7366.882,E2 7366.882} C_VEL
LIN {X 0,Y 465.268,Z 685.03,A -85,B 0,C 180,E1 7372.675,E2 7372.675} C_VEL
LIN {X 0,Y 465.409,Z 685.03,A -85,B 0,C 180,E1 7378.146,E2 7378.146} C_VEL
LIN {X 0,Y 465.399,Z 685.03,A -85,B 0,C 180,E1 7383.722,E2 7383.722} C_VEL
LIN {X 0,Y 465.153,Z 685.03,A -85,B 0,C 180,E1 7389.338,E2 7389.338} C_VEL
LIN {X 0,Y 465.013,Z 685.03,A -85,B 0,C 180,E1 7395.05,E2 7395.05} C_VEL
LIN {X 0,Y 464.909,Z 685.03,A -85,B 0,C 180,E1 7400.921,E2 7400.921} C_VEL
LIN {X 0,Y 464.67,Z 685.03,A -85,B 0,C 180,E1 7407.044,E2 7407.044} C_VEL
LIN {X 0,Y 464.597,Z 685.03,A -85,B 0,C 180,E1 7413.517,E2 7413.517} C_VEL
LIN {X 0,Y 464.603,Z 685.03,A -85,B 0,C 180,E1 7418.786,E2 7418.786} C_VEL
LIN {X 0,Y 464.542,Z 685.03,A -85,B 0,C 180,E1 7424.387,E2 7424.387} C_VEL
LIN {X 0,Y 464.643,Z 685.832,A -85,B 0,C 180,E1 7428.635,E2 7428.635} C_VEL
LIN {X 0,Y 476.638,Z 720.502,A -85,B 0,C 180,E1 7431.925,E2 7431.925} C_VEL
LIN {X 0,Y 487.292,Z 736.475,A -85,B 0,C 180,E1 7433.04,E2 7433.04} C_VEL
LIN {X 0,Y 486.042,Z 778.925,A -85,B 0,C 180,E1 7433.936,E2 7433.936} C_VEL
LIN {X 0,Y 481.514,Z 795.657,A -85,B 0,C 180,E1 7434.245,E2 7434.245} C_VEL
LIN {X 0,Y 477.126,Z 810.064,A -85,B 0,C 180,E1 7434.603,E2 7434.603} C_VEL
LIN {X 0,Y 476.893,Z 812.12,A -85,B 0,C 180,E1 7434.689,E2 7434.689} C_VEL
LIN {X 0,Y 473.349,Z 851.616,A -85,B 0,C 180,E1 7436.86,E2 7436.86} C_VEL
LIN {X 0,Y 469.463,Z 889.33,A -85,B 0,C 180,E1 7439.796,E2 7439.796} C_VEL
LIN {X 0,Y 465.775,Z 922.569,A -85,B 0,C 180,E1 7443.289,E2 7443.289} C_VEL
LIN {X 0,Y 462.964,Z 946.807,A -85,B 0,C 180,E1 7446.638,E2 7446.638} C_VEL
LIN {X 0,Y 460.28,Z 970.812,A -85,B 0,C 180,E1 7451.22,E2 7451.22} C_VEL
LIN {X 0,Y 458.654,Z 989.604,A -85,B 0,C 180,E1 7456.215,E2 7456.215} C_VEL
LIN {X 0,Y 458.032,Z 1000.723,A -85,B 0,C 180,E1 7460.521,E2 7460.521} C_VEL
LIN {X 0,Y 457.748,Z 1006.998,A -85,B 0,C 180,E1 7464.327,E2 7464.327} C_VEL
LIN {X 0,Y 457.715,Z 1010.109,A -85,B 0,C 180,E1 7468.113,E2 7468.113} C_VEL
LIN {X 0,Y 457.772,Z 1010.107,A -85,B 0,C 180,E1 7471.892,E2 7471.892} C_VEL
LIN {X 0,Y 457.849,Z 1005.732,A -85,B 0,C 180,E1 7476.627,E2 7476.627} C_VEL
LIN {X 0,Y 458.198,Z 996.309,A -85,B 0,C 180,E1 7481.4,E2 7481.4} C_VEL
LIN {X 0,Y 459.336,Z 981.285,A -85,B 0,C 180,E1 7486.219,E2 7486.219} C_VEL
LIN {X 0,Y 461.327,Z 960.898,A -85,B 0,C 180,E1 7490.842,E2 7490.842} C_VEL
LIN {X 0,Y 464.124,Z 937.414,A -85,B 0,C 180,E1 7494.788,E2 7494.788} C_VEL
LIN {X 0,Y 467.249,Z 907.413,A -85,B 0,C 180,E1 7498.321,E2 7498.321} C_VEL
LIN {X 0,Y 470.74,Z 871.567,A -85,B 0,C 180,E1 7501.459,E2 7501.459} C_VEL
LIN {X 0,Y 474.024,Z 832.69,A -85,B 0,C 180,E1 7503.931,E2 7503.931} C_VEL
LIN {X 0,Y 476.749,Z 790.598,A -85,B 0,C 180,E1 7505.749,E2 7505.749} C_VEL
LIN {X 0,Y 478.743,Z 745.974,A -85,B 0,C 180,E1 7506.855,E2 7506.855} C_VEL
LIN {X 0,Y 477.952,Z 737.668,A -85,B 0,C 180,E1 7507.049,E2 7507.049} C_VEL
LIN {X 0,Y 466.136,Z 717.525,A -85,B 0,C 180,E1 7508.194,E2 7508.194} C_VEL
LIN {X 0,Y 462.482,Z 706.382,A -85,B 0,C 180,E1 7508.904,E2 7508.904} C_VEL
LIN {X 0,Y 456.644,Z 685.03,A -85,B 0,C 180,E1 7510.806,E2 7510.806} C_VEL
LIN {X 0,Y 456.696,Z 685.03,A -85,B 0,C 180,E1 7516.636,E2 7516.636} C_VEL
LIN {X 0,Y 456.654,Z 685.03,A -85,B 0,C 180,E1 7523.5,E2 7523.5} C_VEL
LIN {X 0,Y 456.666,Z 685.03,A -85,B 0,C 180,E1 7530.285,E2 7530.285} C_VEL
LIN {X 0,Y 456.87,Z 685.03,A -85,B 0,C 180,E1 7536.647,E2 7536.647} C_VEL
LIN {X 0,Y 456.98,Z 685.03,A -85,B 0,C 180,E1 7537.831,E2 7537.831} C_VEL
LIN {X 0,Y 467.455,Z 714.52,A -85,B 0,C 180,E1 7539.621,E2 7539.621} C_VEL
LIN {X 0,Y 465.946,Z 765.679,A -85,B 0,C 180,E1 7541.047,E2 7541.047} C_VEL
LIN {X 0,Y 464.88,Z 792.876,A -85,B 0,C 180,E1 7542.524,E2 7542.524} C_VEL
LIN {X 0,Y 463.271,Z 817.352,A -85,B 0,C 180,E1 7544.651,E2 7544.651} C_VEL
LIN {X 0,Y 461.776,Z 837.498,A -85,B 0,C 180,E1 7547.254,E2 7547.254} C_VEL
LIN {X 0,Y 460.483,Z 852.752,A -85,B 0,C 180,E1 7550.14,E2 7550.14} C_VEL
LIN {X 0,Y 459.596,Z 863.878,A -85,B 0,C 180,E1 7553.398,E2 7553.398} C_VEL
LIN {X 0,Y 459.154,Z 869.409,A -85,B 0,C 180,E1 7556.227,E2 7556.227} C_VEL
LIN {X 0,Y 458.968,Z 871.647,A -85,B 0,C 180,E1 7559.996,E2 7559.996} C_VEL
LIN {X 0,Y 458.979,Z 868.097,A -85,B 0,C 180,E1 7563.766,E2 7563.766} C_VEL
LIN {X 0,Y 459.342,Z 858.486,A -85,B 0,C 180,E1 7567.546,E2 7567.546} C_VEL
LIN {X 0,Y 460.217,Z 843.437,A -85,B 0,C 180,E1 7570.947,E2 7570.947} C_VEL
LIN {X 0,Y 461.545,Z 823.224,A -85,B 0,C 180,E1 7573.947,E2 7573.947} C_VEL
LIN {X 0,Y 462.95,Z 799.197,A -85,B 0,C 180,E1 7576.348,E2 7576.348} C_VEL
LIN {X 0,Y 464.347,Z 771.134,A -85,B 0,C 180,E1 7578.16,E2 7578.16} C_VEL
LIN {X 0,Y 465.112,Z 741.996,A -85,B 0,C 180,E1 7579.224,E2 7579.224} C_VEL
LIN {X 0,Y 464.895,Z 710.682,A -85,B 0,C 180,E1 7579.863,E2 7579.863} C_VEL
LIN {X 0,Y 457.033,Z 685.03,A -85,B 0,C 180,E1 7580.82,E2 7580.82} C_VEL
LIN {X 0,Y 456.766,Z 685.03,A -85,B 0,C 180,E1 7587.542,E2 7587.542} C_VEL
LIN {X 0,Y 456.656,Z 685.03,A -85,B 0,C 180,E1 7594.289,E2 7594.289} C_VEL
LIN {X 0,Y 456.662,Z 685.03,A -85,B 0,C 180,E1 7600.526,E2 7600.526} C_VEL
LIN {X 0,Y 456.675,Z 685.03,A -85,B 0,C 180,E1 7606.62,E2 7606.62} C_VEL
LIN {X 0,Y 456.663,Z 685.03,A -85,B 0,C 180,E1 7613.496,E2 7613.496} C_VEL
LIN {X 0,Y 456.732,Z 685.03,A -85,B 0,C 180,E1 7620.287,E2 7620.287} C_VEL
LIN {X 0,Y 456.877,Z 685.03,A -85,B 0,C 180,E1 7622.348,E2 7622.348} C_VEL
LIN {X 0,Y 469.127,Z 719.945,A -85,B 0,C 180,E1 7624.158,E2 7624.158} C_VEL
LIN {X 0,Y 469.695,Z 732.865,A -85,B 0,C 180,E1 7624.781,E2 7624.781} C_VEL
LIN {X 0,Y 467.638,Z 764.535,A -85,B 0,C 180,E1 7626.677,E2 7626.677} C_VEL
LIN {X 0,Y 465.178,Z 793.04,A -85,B 0,C 180,E1 7629.217,E2 7629.217} C_VEL
LIN {X 0,Y 462.803,Z 816.722,A -85,B 0,C 180,E1 7632.197,E2 7632.197} C_VEL
LIN {X 0,Y 460.691,Z 837.269,A -85,B 0,C 180,E1 7635.84,E2 7635.84} C_VEL
LIN {X 0,Y 459.384,Z 851.893,A -85,B 0,C 180,E1 7639.589,E2 7639.589} C_VEL
LIN {X 0,Y 458.675,Z 861.413,A -85,B 0,C 180,E1 7643.385,E2 7643.385} C_VEL
LIN {X 0,Y 458.484,Z 865.625,A -85,B 0,C 180,E1 7646.223,E2 7646.223} C_VEL
LIN {X 0,Y 458.407,Z 867.606,A -85,B 0,C 180,E1 7649.997,E2 7649.997} C_VEL
LIN {X 0,Y 458.564,Z 864.395,A -85,B 0,C 180,E1 7654.716,E2 7654.716} C_VEL
LIN {X 0,Y 459.114,Z 855.781,A -85,B 0,C 180,E1 7658.979,E2 7658.979} C_VEL
LIN {X 0,Y 460.314,Z 841.908,A -85,B 0,C 180,E1 7663.023,E2 7663.023} C_VEL
LIN {X 0,Y 462.253,Z 822.328,A -85,B 0,C 180,E1 7666.839,E2 7666.839} C_VEL
LIN {X 0,Y 464.546,Z 799.041,A -85,B 0,C 180,E1 7670.033,E2 7670.033} C_VEL
LIN {X 0,Y 467.069,Z 771.631,A -85,B 0,C 180,E1 7672.684,E2 7672.684} C_VEL
LIN {X 0,Y 469.173,Z 741.165,A -85,B 0,C 180,E1 7674.714,E2 7674.714} C_VEL
LIN {X 0,Y 469.549,Z 720.854,A -85,B 0,C 180,E1 7675.684,E2 7675.684} C_VEL
LIN {X 0,Y 457.746,Z 688.758,A -85,B 0,C 180,E1 7677.414,E2 7677.414} C_VEL
LIN {X 0,Y 456.802,Z 685.03,A -85,B 0,C 180,E1 7677.545,E2 7677.545} C_VEL
LIN {X 0,Y 456.663,Z 685.03,A -85,B 0,C 180,E1 7684.314,E2 7684.314} C_VEL
LIN {X 0,Y 456.576,Z 685.03,A -85,B 0,C 180,E1 7690.534,E2 7690.534} C_VEL
LIN {X 0,Y 456.649,Z 685.03,A -85,B 0,C 180,E1 7696.634,E2 7696.634} C_VEL
LIN {X 0,Y 456.667,Z 685.03,A -85,B 0,C 180,E1 7702.471,E2 7702.471} C_VEL
LIN {X 0,Y 456.672,Z 685.03,A -85,B 0,C 180,E1 7709.218,E2 7709.218} C_VEL
LIN {X 0,Y 456.829,Z 685.03,A -85,B 0,C 180,E1 7714.576,E2 7714.576} C_VEL
LIN {X 0,Y 457.074,Z 685.03,A -85,B 0,C 180,E1 7720.729,E2 7720.729} C_VEL
LIN {X 0,Y 457.319,Z 685.03,A -85,B 0,C 180,E1 7726.651,E2 7726.651} C_VEL
LIN {X 0,Y 457.344,Z 685.03,A -85,B 0,C 180,E1 7732.667,E2 7732.667} C_VEL
LIN {X 0,Y 457.506,Z 685.03,A -85,B 0,C 180,E1 7738.114,E2 7738.114} C_VEL
LIN {X 0,Y 457.489,Z 685.03,A -85,B 0,C 180,E1 7743.786,E2 7743.786} C_VEL
LIN {X 0,Y 457.249,Z 685.03,A -85,B 0,C 180,E1 7749.501,E2 7749.501} C_VEL
LIN {X 0,Y 457.079,Z 685.03,A -85,B 0,C 180,E1 7755.317,E2 7755.317} C_VEL
LIN {X 0,Y 456.948,Z 685.03,A -85,B 0,C 180,E1 7761.303,E2 7761.303} C_VEL
LIN {X 0,Y 456.743,Z 685.03,A -85,B 0,C 180,E1 7767.553,E2 7767.553} C_VEL
LIN {X 0,Y 456.64,Z 685.03,A -85,B 0,C 180,E1 7774.296,E2 7774.296} C_VEL
LIN {X 0,Y 456.689,Z 685.03,A -85,B 0,C 180,E1 7780.539,E2 7780.539} C_VEL
LIN {X 0,Y 456.634,Z 685.03,A -85,B 0,C 180,E1 7787.098,E2 7787.098} C_VEL
LIN {X 0,Y 456.67,Z 685.679,A -85,B 0,C 180,E1 7787.927,E2 7787.927} C_VEL
LIN {X 0,Y 468.365,Z 719.604,A -85,B 0,C 180,E1 7791.237,E2 7791.237} C_VEL
LIN {X 0,Y 480.549,Z 739.893,A -85,B 0,C 180,E1 7792.595,E2 7792.595} C_VEL
LIN {X 0,Y 479,Z 782.728,A -85,B 0,C 180,E1 7793.582,E2 7793.582} C_VEL
LIN {X 0,Y 476.893,Z 812.12,A -85,B 0,C 180,E1 7794.689,E2 7794.689} C_VEL
LIN {X 0,Y 471.919,Z 828.345,A -85,B 0,C 180,E1 7795.255,E2 7795.255} C_VEL
LIN {X 0,Y 467.197,Z 842.148,A -85,B 0,C 180,E1 7795.841,E2 7795.841} C_VEL
LIN {X 0,Y 466.958,Z 844.086,A -85,B 0,C 180,E1 7795.961,E2 7795.961} C_VEL
LIN {X 0,Y 462.963,Z 881.429,A -85,B 0,C 180,E1 7798.74,E2 7798.74} C_VEL
LIN {X 0,Y 458.979,Z 915.7,A -85,B 0,C 180,E1 7802.198,E2 7802.198} C_VEL
LIN {X 0,Y 455.368,Z 945.985,A -85,B 0,C 180,E1 7806.27,E2 7806.27} C_VEL
LIN {X 0,Y 453.017,Z 967.023,A -85,B 0,C 180,E1 7810.052,E2 7810.052} C_VEL
LIN {X 0,Y 451.117,Z 986.313,A -85,B 0,C 180,E1 7814.935,E2 7814.935} C_VEL
LIN {X 0,Y 450.227,Z 999.712,A -85,B 0,C 180,E1 7819.868,E2 7819.868} C_VEL
LIN {X 0,Y 449.87,Z 1006.999,A -85,B 0,C 180,E1 7824.227,E2 7824.227} C_VEL
LIN {X 0,Y 449.834,Z 1010.107,A -85,B 0,C 180,E1 7828.08,E2 7828.08} C_VEL
LIN {X 0,Y 449.885,Z 1010.106,A -85,B 0,C 180,E1 7831.925,E2 7831.925} C_VEL
LIN {X 0,Y 449.944,Z 1005.731,A -85,B 0,C 180,E1 7836.744,E2 7836.744} C_VEL
LIN {X 0,Y 450.345,Z 996.308,A -85,B 0,C 180,E1 7841.602,E2 7841.602} C_VEL
LIN {X 0,Y 451.574,Z 981.284,A -85,B 0,C 180,E1 7846.505,E2 7846.505} C_VEL
LIN {X 0,Y 453.771,Z 960.543,A -85,B 0,C 180,E1 7851.259,E2 7851.259} C_VEL
LIN {X 0,Y 456.374,Z 936.787,A -85,B 0,C 180,E1 7855.015,E2 7855.015} C_VEL
LIN {X 0,Y 459.833,Z 904.522,A -85,B 0,C 180,E1 7858.82,E2 7858.82} C_VEL
LIN {X 0,Y 463.462,Z 868.205,A -85,B 0,C 180,E1 7861.985,E2 7861.985} C_VEL
LIN {X 0,Y 466.85,Z 829.116,A -85,B 0,C 180,E1 7864.452,E2 7864.452} C_VEL
LIN {X 0,Y 469.75,Z 786.743,A -85,B 0,C 180,E1 7866.263,E2 7866.263} C_VEL
LIN {X 0,Y 471.789,Z 743.027,A -85,B 0,C 180,E1 7867.339,E2 7867.339} C_VEL
LIN {X 0,Y 458.354,Z 717.394,A -85,B 0,C 180,E1 7868.784,E2 7868.784} C_VEL
LIN {X 0,Y 454.733,Z 705.699,A -85,B 0,C 180,E1 7869.492,E2 7869.492} C_VEL
LIN {X 0,Y 448.7,Z 685.03,A -85,B 0,C 180,E1 7871.492,E2 7871.492} C_VEL
LIN {X 0,Y 448.743,Z 685.03,A -85,B 0,C 180,E1 7877.735,E2 7877.735} C_VEL
LIN {X 0,Y 448.711,Z 685.03,A -85,B 0,C 180,E1 7883.824,E2 7883.824} C_VEL
LIN {X 0,Y 448.73,Z 685.03,A -85,B 0,C 180,E1 7889.705,E2 7889.705} C_VEL
LIN {X 0,Y 448.988,Z 685.03,A -85,B 0,C 180,E1 7896.717,E2 7896.717} C_VEL
LIN {X 0,Y 448.985,Z 685.251,A -85,B 0,C 180,E1 7897.094,E2 7897.094} C_VEL
LIN {X 0,Y 460.151,Z 715.009,A -85,B 0,C 180,E1 7899.122,E2 7899.122} C_VEL
LIN {X 0,Y 458.69,Z 769.935,A -85,B 0,C 180,E1 7900.79,E2 7900.79} C_VEL
LIN {X 0,Y 457.358,Z 798.272,A -85,B 0,C 180,E1 7902.475,E2 7902.475} C_VEL
LIN {X 0,Y 455.617,Z 822.458,A -85,B 0,C 180,E1 7904.755,E2 7904.755} C_VEL
LIN {X 0,Y 453.84,Z 843.503,A -85,B 0,C 180,E1 7907.759,E2 7907.759} C_VEL
LIN {X 0,Y 452.53,Z 857.939,A -85,B 0,C 180,E1 7910.883,E2 7910.883} C_VEL
LIN {X 0,Y 451.644,Z 867.597,A -85,B 0,C 180,E1 7914.244,E2 7914.244} C_VEL
LIN {X 0,Y 451.234,Z 872.641,A -85,B 0,C 180,E1 7918.079,E2 7918.079} C_VEL
LIN {X 0,Y 451.134,Z 871.913,A -85,B 0,C 180,E1 7921.912,E2 7921.912} C_VEL
LIN {X 0,Y 451.361,Z 865.315,A -85,B 0,C 180,E1 7925.751,E2 7925.751} C_VEL
LIN {X 0,Y 451.989,Z 853.149,A -85,B 0,C 180,E1 7929.362,E2 7929.362} C_VEL
LIN {X 0,Y 453.163,Z 836.421,A -85,B 0,C 180,E1 7932.495,E2 7932.495} C_VEL
LIN {X 0,Y 454.628,Z 814.602,A -85,B 0,C 180,E1 7935.27,E2 7935.27} C_VEL
LIN {X 0,Y 456.074,Z 789.25,A -85,B 0,C 180,E1 7937.443,E2 7937.443} C_VEL
LIN {X 0,Y 457.279,Z 761.234,A -85,B 0,C 180,E1 7938.95,E2 7938.95} C_VEL
LIN {X 0,Y 457.853,Z 729.348,A -85,B 0,C 180,E1 7939.828,E2 7939.828} C_VEL
LIN {X 0,Y 457.45,Z 712.138,A -85,B 0,C 180,E1 7940.196,E2 7940.196} C_VEL
LIN {X 0,Y 449.106,Z 685.03,A -85,B 0,C 180,E1 7941.215,E2 7941.215} C_VEL
LIN {X 0,Y 448.776,Z 685.03,A -85,B 0,C 180,E1 7948.075,E2 7948.075} C_VEL
LIN {X 0,Y 448.708,Z 685.03,A -85,B 0,C 180,E1 7954.861,E2 7954.861} C_VEL
LIN {X 0,Y 448.743,Z 685.03,A -85,B 0,C 180,E1 7959.702,E2 7959.702} C_VEL
LIN {X 0,Y 448.676,Z 685.03,A -85,B 0,C 180,E1 7965.06,E2 7965.06} C_VEL
LIN {X 0,Y 448.754,Z 685.03,A -85,B 0,C 180,E1 7970.648,E2 7970.648} C_VEL
LIN {X 0,Y 448.7,Z 685.03,A -85,B 0,C 180,E1 7977.441,E2 7977.441} C_VEL
LIN {X 0,Y 448.979,Z 685.03,A -85,B 0,C 180,E1 7981.801,E2 7981.801} C_VEL
LIN {X 0,Y 461.509,Z 720.018,A -85,B 0,C 180,E1 7983.648,E2 7983.648} C_VEL
LIN {X 0,Y 462.87,Z 729.38,A -85,B 0,C 180,E1 7984.153,E2 7984.153} C_VEL
LIN {X 0,Y 460.841,Z 761.315,A -85,B 0,C 180,E1 7985.964,E2 7985.964} C_VEL
LIN {X 0,Y 458.342,Z 789.61,A -85,B 0,C 180,E1 7988.383,E2 7988.383} C_VEL
LIN {X 0,Y 455.701,Z 814.656,A -85,B 0,C 180,E1 7991.41,E2 7991.41} C_VEL
LIN {X 0,Y 453.359,Z 836.016,A -85,B 0,C 180,E1 7995.059,E2 7995.059} C_VEL
LIN {X 0,Y 451.866,Z 851.55,A -85,B 0,C 180,E1 7998.926,E2 7998.926} C_VEL
LIN {X 0,Y 450.937,Z 862.656,A -85,B 0,C 180,E1 8003.271,E2 8003.271} C_VEL
LIN {X 0,Y 450.696,Z 866.872,A -85,B 0,C 180,E1 8006.157,E2 8006.157} C_VEL
LIN {X 0,Y 450.619,Z 868.851,A -85,B 0,C 180,E1 8009.997,E2 8009.997} C_VEL
LIN {X 0,Y 450.781,Z 865.644,A -85,B 0,C 180,E1 8014.798,E2 8014.798} C_VEL
LIN {X 0,Y 451.383,Z 857.088,A -85,B 0,C 180,E1 8019.112,E2 8019.112} C_VEL
LIN {X 0,Y 452.698,Z 843.157,A -85,B 0,C 180,E1 8023.246,E2 8023.246} C_VEL
LIN {X 0,Y 454.62,Z 825.07,A -85,B 0,C 180,E1 8026.882,E2 8026.882} C_VEL
LIN {X 0,Y 457.055,Z 801.92,A -85,B 0,C 180,E1 8030.167,E2 8030.167} C_VEL
LIN {X 0,Y 459.766,Z 774.204,A -85,B 0,C 180,E1 8032.947,E2 8032.947} C_VEL
LIN {X 0,Y 462.04,Z 743.532,A -85,B 0,C 180,E1 8035.057,E2 8035.057} C_VEL
LIN {X 0,Y 462.447,Z 722.886,A -85,B 0,C 180,E1 8036.074,E2 8036.074} C_VEL
LIN {X 0,Y 450.576,Z 690.247,A -85,B 0,C 180,E1 8037.882,E2 8037.882} C_VEL
LIN {X 0,Y 448.823,Z 685.03,A -85,B 0,C 180,E1 8038.2,E2 8038.2} C_VEL
LIN {X 0,Y 448.701,Z 685.03,A -85,B 0,C 180,E1 8044.869,E2 8044.869} C_VEL
LIN {X 0,Y 448.656,Z 685.03,A -85,B 0,C 180,E1 8049.719,E2 8049.719} C_VEL
LIN {X 0,Y 448.643,Z 685.03,A -85,B 0,C 180,E1 8055.074,E2 8055.074} C_VEL
LIN {X 0,Y 448.744,Z 685.03,A -85,B 0,C 180,E1 8060.662,E2 8060.662} C_VEL
LIN {X 0,Y 448.699,Z 685.03,A -85,B 0,C 180,E1 8067.455,E2 8067.455} C_VEL
LIN {X 0,Y 448.911,Z 685.03,A -85,B 0,C 180,E1 8074.095,E2 8074.095} C_VEL
LIN {X 0,Y 449.118,Z 685.03,A -85,B 0,C 180,E1 8080.373,E2 8080.373} C_VEL
LIN {X 0,Y 449.394,Z 685.03,A -85,B 0,C 180,E1 8086.85,E2 8086.85} C_VEL
LIN {X 0,Y 449.433,Z 685.03,A -85,B 0,C 180,E1 8092.662,E2 8092.662} C_VEL
LIN {X 0,Y 449.621,Z 685.03,A -85,B 0,C 180,E1 8098.081,E2 8098.081} C_VEL
LIN {X 0,Y 449.579,Z 685.03,A -85,B 0,C 180,E1 8103.853,E2 8103.853} C_VEL
LIN {X 0,Y 449.324,Z 685.03,A -85,B 0,C 180,E1 8109.67,E2 8109.67} C_VEL
LIN {X 0,Y 449.157,Z 685.03,A -85,B 0,C 180,E1 8115.594,E2 8115.594} C_VEL
LIN {X 0,Y 449.016,Z 685.03,A -85,B 0,C 180,E1 8121.698,E2 8121.698} C_VEL
LIN {X 0,Y 448.757,Z 685.03,A -85,B 0,C 180,E1 8128.086,E2 8128.086} C_VEL
LIN {X 0,Y 448.695,Z 685.03,A -85,B 0,C 180,E1 8134.872,E2 8134.872} C_VEL
LIN {X 0,Y 448.757,Z 685.03,A -85,B 0,C 180,E1 8139.711,E2 8139.711} C_VEL
LIN {X 0,Y 448.701,Z 685.03,A -85,B 0,C 180,E1 8146.041,E2 8146.041} C_VEL
LIN {X 0,Y 448.762,Z 685.139,A -85,B 0,C 180,E1 8147.177,E2 8147.177} C_VEL
LIN {X 0,Y 460.364,Z 718.827,A -85,B 0,C 180,E1 8150.544,E2 8150.544} C_VEL
LIN {X 0,Y 471.603,Z 739.912,A -85,B 0,C 180,E1 8151.902,E2 8151.902} C_VEL
LIN {X 0,Y 473.925,Z 743.3,A -85,B 0,C 180,E1 8152.144,E2 8152.144} C_VEL
LIN {X 0,Y 471.966,Z 786.042,A -85,B 0,C 180,E1 8153.197,E2 8153.197} C_VEL
LIN {X 0,Y 468.713,Z 826.771,A -85,B 0,C 180,E1 8154.957,E2 8154.957} C_VEL
LIN {X 0,Y 466.958,Z 844.086,A -85,B 0,C 180,E1 8155.961,E2 8155.961} C_VEL
LIN {X 0,Y 465.138,Z 851.917,A -85,B 0,C 180,E1 8156.41,E2 8156.41} C_VEL
LIN {X 0,Y 456.786,Z 872.459,A -85,B 0,C 180,E1 8157.6,E2 8157.6} C_VEL
LIN {X 0,Y 456.475,Z 874.284,A -85,B 0,C 180,E1 8157.748,E2 8157.748} C_VEL
LIN {X 0,Y 452.076,Z 909.6,A -85,B 0,C 180,E1 8161.191,E2 8161.191} C_VEL
LIN {X 0,Y 448.318,Z 940.066,A -85,B 0,C 180,E1 8165.16,E2 8165.16} C_VEL
LIN {X 0,Y 445.259,Z 966.355,A -85,B 0,C 180,E1 8169.731,E2 8169.731} C_VEL
LIN {X 0,Y 443.54,Z 983.085,A -85,B 0,C 180,E1 8173.701,E2 8173.701} C_VEL
LIN {X 0,Y 442.458,Z 997.508,A -85,B 0,C 180,E1 8178.693,E2 8178.693} C_VEL
LIN {X 0,Y 442.084,Z 1005.737,A -85,B 0,C 180,E1 8183.141,E2 8183.141} C_VEL
LIN {X 0,Y 441.928,Z 1010.106,A -85,B 0,C 180,E1 8188.046,E2 8188.046} C_VEL
LIN {X 0,Y 441.979,Z 1010.103,A -85,B 0,C 180,E1 8191.96,E2 8191.96} C_VEL
LIN {X 0,Y 442.076,Z 1005.73,A -85,B 0,C 180,E1 8196.865,E2 8196.865} C_VEL
LIN {X 0,Y 442.494,Z 996.307,A -85,B 0,C 180,E1 8201.811,E2 8201.811} C_VEL
LIN {X 0,Y 443.843,Z 981.283,A -85,B 0,C 180,E1 8206.801,E2 8206.801} C_VEL
LIN {X 0,Y 445.561,Z 963.791,A -85,B 0,C 180,E1 8210.732,E2 8210.732} C_VEL
LIN {X 0,Y 448.413,Z 937.81,A -85,B 0,C 180,E1 8214.991,E2 8214.991} C_VEL
LIN {X 0,Y 451.775,Z 907.682,A -85,B 0,C 180,E1 8218.7,E2 8218.7} C_VEL
LIN {X 0,Y 455.381,Z 873.402,A -85,B 0,C 180,E1 8221.87,E2 8221.87} C_VEL
LIN {X 0,Y 459.027,Z 834.668,A -85,B 0,C 180,E1 8224.493,E2 8224.493} C_VEL
LIN {X 0,Y 462.192,Z 792.669,A -85,B 0,C 180,E1 8226.463,E2 8226.463} C_VEL
LIN {X 0,Y 464.685,Z 748.851,A -85,B 0,C 180,E1 8227.69,E2 8227.69} C_VEL
LIN {X 0,Y 463.9,Z 743.62,A -85,B 0,C 180,E1 8227.853,E2 8227.853} C_VEL
LIN {X 0,Y 452.713,Z 722.318,A -85,B 0,C 180,E1 8229.138,E2 8229.138} C_VEL
LIN {X 0,Y 446.944,Z 704.91,A -85,B 0,C 180,E1 8230.147,E2 8230.147} C_VEL
LIN {X 0,Y 440.779,Z 685.03,A -85,B 0,C 180,E1 8232.243,E2 8232.243} C_VEL
LIN {X 0,Y 440.753,Z 685.03,A -85,B 0,C 180,E1 8239.419,E2 8239.419} C_VEL
LIN {X 0,Y 440.792,Z 685.03,A -85,B 0,C 180,E1 8245.256,E2 8245.256} C_VEL
LIN {X 0,Y 440.873,Z 685.03,A -85,B 0,C 180,E1 8251.365,E2 8251.365} C_VEL
LIN {X 0,Y 441.04,Z 685.468,A -85,B 0,C 180,E1 8256.259,E2 8256.259} C_VEL
LIN {X 0,Y 451.701,Z 711.942,A -85,B 0,C 180,E1 8258.36,E2 8258.36} C_VEL
LIN {X 0,Y 453.476,Z 719.775,A -85,B 0,C 180,E1 8258.773,E2 8258.773} C_VEL
LIN {X 0,Y 451.572,Z 769.865,A -85,B 0,C 180,E1 8260.337,E2 8260.337} C_VEL
LIN {X 0,Y 450.316,Z 797.37,A -85,B 0,C 180,E1 8261.94,E2 8261.94} C_VEL
LIN {X 0,Y 448.474,Z 821.58,A -85,B 0,C 180,E1 8264.179,E2 8264.179} C_VEL
LIN {X 0,Y 446.615,Z 842.407,A -85,B 0,C 180,E1 8267.062,E2 8267.062} C_VEL
LIN {X 0,Y 445.068,Z 857.676,A -85,B 0,C 180,E1 8270.236,E2 8270.236} C_VEL
LIN {X 0,Y 444.082,Z 868.031,A -85,B 0,C 180,E1 8273.656,E2 8273.656} C_VEL
LIN {X 0,Y 443.699,Z 872.29,A -85,B 0,C 180,E1 8276.096,E2 8276.096} C_VEL
LIN {X 0,Y 443.428,Z 874.361,A -85,B 0,C 180,E1 8279.996,E2 8279.996} C_VEL
LIN {X 0,Y 443.451,Z 870.619,A -85,B 0,C 180,E1 8283.898,E2 8283.898} C_VEL
LIN {X 0,Y 443.874,Z 860.811,A -85,B 0,C 180,E1 8287.811,E2 8287.811} C_VEL
LIN {X 0,Y 444.825,Z 846.024,A -85,B 0,C 180,E1 8291.242,E2 8291.242} C_VEL
LIN {X 0,Y 446.232,Z 827.035,A -85,B 0,C 180,E1 8294.186,E2 8294.186} C_VEL
LIN {X 0,Y 447.838,Z 802.686,A -85,B 0,C 180,E1 8296.763,E2 8296.763} C_VEL
LIN {X 0,Y 449.322,Z 774.981,A -85,B 0,C 180,E1 8298.663,E2 8298.663} C_VEL
LIN {X 0,Y 450.28,Z 745.14,A -85,B 0,C 180,E1 8299.838,E2 8299.838} C_VEL
LIN {X 0,Y 450.143,Z 713.856,A -85,B 0,C 180,E1 8300.524,E2 8300.524} C_VEL
LIN {X 0,Y 441.149,Z 685.03,A -85,B 0,C 180,E1 8301.629,E2 8301.629} C_VEL
LIN {X 0,Y 440.857,Z 685.03,A -85,B 0,C 180,E1 8308.626,E2 8308.626} C_VEL
LIN {X 0,Y 440.804,Z 685.03,A -85,B 0,C 180,E1 8315.58,E2 8315.58} C_VEL
LIN {X 0,Y 440.736,Z 685.03,A -85,B 0,C 180,E1 8321.12,E2 8321.12} C_VEL
LIN {X 0,Y 440.717,Z 685.03,A -85,B 0,C 180,E1 8326.774,E2 8326.774} C_VEL
LIN {X 0,Y 440.795,Z 685.03,A -85,B 0,C 180,E1 8331.954,E2 8331.954} C_VEL
LIN {X 0,Y 440.772,Z 685.03,A -85,B 0,C 180,E1 8338.841,E2 8338.841} C_VEL
LIN {X 0,Y 441.033,Z 685.03,A -85,B 0,C 180,E1 8341.226,E2 8341.226} C_VEL
LIN {X 0,Y 453.847,Z 720.083,A -85,B 0,C 180,E1 8343.115,E2 8343.115} C_VEL
LIN {X 0,Y 455.839,Z 730.913,A -85,B 0,C 180,E1 8343.741,E2 8343.741} C_VEL
LIN {X 0,Y 453.725,Z 762.515,A -85,B 0,C 180,E1 8345.561,E2 8345.561} C_VEL
LIN {X 0,Y 451.059,Z 791.171,A -85,B 0,C 180,E1 8348.052,E2 8348.052} C_VEL
LIN {X 0,Y 448.302,Z 815.893,A -85,B 0,C 180,E1 8351.092,E2 8351.092} C_VEL
LIN {X 0,Y 445.815,Z 837.258,A -85,B 0,C 180,E1 8354.8,E2 8354.8} C_VEL
LIN {X 0,Y 444.214,Z 852.793,A -85,B 0,C 180,E1 8358.732,E2 8358.732} C_VEL
LIN {X 0,Y 443.179,Z 863.903,A -85,B 0,C 180,E1 8363.152,E2 8363.152} C_VEL
LIN {X 0,Y 442.915,Z 868.118,A -85,B 0,C 180,E1 8366.09,E2 8366.09} C_VEL
LIN {X 0,Y 442.836,Z 870.096,A -85,B 0,C 180,E1 8369.997,E2 8369.997} C_VEL
LIN {X 0,Y 443.001,Z 866.893,A -85,B 0,C 180,E1 8374.882,E2 8374.882} C_VEL
LIN {X 0,Y 443.785,Z 857.436,A -85,B 0,C 180,E1 8379.624,E2 8379.624} C_VEL
LIN {X 0,Y 445.176,Z 843.395,A -85,B 0,C 180,E1 8383.724,E2 8383.724} C_VEL
LIN {X 0,Y 447.527,Z 823.305,A -85,B 0,C 180,E1 8387.664,E2 8387.664} C_VEL
LIN {X 0,Y 450.226,Z 799.109,A -85,B 0,C 180,E1 8390.988,E2 8390.988} C_VEL
LIN {X 0,Y 452.967,Z 770.712,A -85,B 0,C 180,E1 8393.731,E2 8393.731} C_VEL
LIN {X 0,Y 455.34,Z 739.229,A -85,B 0,C 180,E1 8395.768,E2 8395.768} C_VEL
LIN {X 0,Y 455.362,Z 724.852,A -85,B 0,C 180,E1 8396.478,E2 8396.478} C_VEL
LIN {X 0,Y 443.93,Z 693.34,A -85,B 0,C 180,E1 8398.298,E2 8398.298} C_VEL
LIN {X 0,Y 440.883,Z 685.03,A -85,B 0,C 180,E1 8398.745,E2 8398.745} C_VEL
LIN {X 0,Y 440.776,Z 685.03,A -85,B 0,C 180,E1 8405.59,E2 8405.59} C_VEL
LIN {X 0,Y 440.66,Z 685.03,A -85,B 0,C 180,E1 8411.129,E2 8411.129} C_VEL
LIN {X 0,Y 440.689,Z 685.03,A -85,B 0,C 180,E1 8416.788,E2 8416.788} C_VEL
LIN {X 0,Y 440.783,Z 685.03,A -85,B 0,C 180,E1 8421.969,E2 8421.969} C_VEL
LIN {X 0,Y 440.751,Z 685.03,A -85,B 0,C 180,E1 8426.793,E2 8426.793} C_VEL
LIN {X 0,Y 440.933,Z 685.03,A -85,B 0,C 180,E1 8433.591,E2 8433.591} C_VEL
LIN {X 0,Y 441.185,Z 685.03,A -85,B 0,C 180,E1 8440.006,E2 8440.006} C_VEL
LIN {X 0,Y 441.452,Z 685.03,A -85,B 0,C 180,E1 8446.162,E2 8446.162} C_VEL
LIN {X 0,Y 441.542,Z 685.03,A -85,B 0,C 180,E1 8452.655,E2 8452.655} C_VEL
LIN {X 0,Y 441.717,Z 685.03,A -85,B 0,C 180,E1 8458.047,E2 8458.047} C_VEL
LIN {X 0,Y 441.669,Z 685.03,A -85,B 0,C 180,E1 8463.922,E2 8463.922} C_VEL
LIN {X 0,Y 441.428,Z 685.03,A -85,B 0,C 180,E1 8469.845,E2 8469.845} C_VEL
LIN {X 0,Y 441.195,Z 685.03,A -85,B 0,C 180,E1 8476.73,E2 8476.73} C_VEL
LIN {X 0,Y 441.005,Z 685.03,A -85,B 0,C 180,E1 8482.502,E2 8482.502} C_VEL
LIN {X 0,Y 440.843,Z 685.03,A -85,B 0,C 180,E1 8488.637,E2 8488.637} C_VEL
LIN {X 0,Y 440.795,Z 685.03,A -85,B 0,C 180,E1 8495.591,E2 8495.591} C_VEL
LIN {X 0,Y 440.749,Z 685.03,A -85,B 0,C 180,E1 8501.131,E2 8501.131} C_VEL
LIN {X 0,Y 440.801,Z 685.104,A -85,B 0,C 180,E1 8506.441,E2 8506.441} C_VEL
LIN {X 0,Y 452.345,Z 718.156,A -85,B 0,C 180,E1 8509.831,E2 8509.831} C_VEL
LIN {X 0,Y 465.437,Z 743.868,A -85,B 0,C 180,E1 8511.476,E2 8511.476} C_VEL
LIN {X 0,Y 467.184,Z 746.294,A -85,B 0,C 180,E1 8511.666,E2 8511.666} C_VEL
LIN {X 0,Y 464.934,Z 789.209,A -85,B 0,C 180,E1 8512.816,E2 8512.816} C_VEL
LIN {X 0,Y 461.437,Z 829.081,A -85,B 0,C 180,E1 8514.63,E2 8514.63} C_VEL
LIN {X 0,Y 457.468,Z 865.936,A -85,B 0,C 180,E1 8517.079,E2 8517.079} C_VEL
LIN {X 0,Y 456.475,Z 874.284,A -85,B 0,C 180,E1 8517.748,E2 8517.748} C_VEL
LIN {X 0,Y 451.001,Z 888.649,A -85,B 0,C 180,E1 8518.839,E2 8518.839} C_VEL
LIN {X 0,Y 445.578,Z 902.249,A -85,B 0,C 180,E1 8520.049,E2 8520.049} C_VEL
LIN {X 0,Y 441.41,Z 933.524,A -85,B 0,C 180,E1 8523.962,E2 8523.962} C_VEL
LIN {X 0,Y 438.086,Z 960.393,A -85,B 0,C 180,E1 8528.438,E2 8528.438} C_VEL
LIN {X 0,Y 435.934,Z 980.35,A -85,B 0,C 180,E1 8532.894,E2 8532.894} C_VEL
LIN {X 0,Y 434.709,Z 995.261,A -85,B 0,C 180,E1 8537.546,E2 8537.546} C_VEL
LIN {X 0,Y 434.214,Z 1004.269,A -85,B 0,C 180,E1 8542.012,E2 8542.012} C_VEL
LIN {X 0,Y 434.006,Z 1008.94,A -85,B 0,C 180,E1 8546.015,E2 8546.015} C_VEL
LIN {X 0,Y 434.035,Z 1010.5,A -85,B 0,C 180,E1 8550.003,E2 8550.003} C_VEL
LIN {X 0,Y 434.018,Z 1008.92,A -85,B 0,C 180,E1 8553.991,E2 8553.991} C_VEL
LIN {X 0,Y 434.295,Z 1002.588,A -85,B 0,C 180,E1 8558.999,E2 8558.999} C_VEL
LIN {X 0,Y 435.087,Z 990.859,A -85,B 0,C 180,E1 8564.054,E2 8564.054} C_VEL
LIN {X 0,Y 436.6,Z 973.771,A -85,B 0,C 180,E1 8568.649,E2 8568.649} C_VEL
LIN {X 0,Y 439.224,Z 949.772,A -85,B 0,C 180,E1 8573.276,E2 8573.276} C_VEL
LIN {X 0,Y 442.502,Z 921.603,A -85,B 0,C 180,E1 8577.302,E2 8577.302} C_VEL
LIN {X 0,Y 446.268,Z 887.923,A -85,B 0,C 180,E1 8580.906,E2 8580.906} C_VEL
LIN {X 0,Y 450.251,Z 850.076,A -85,B 0,C 180,E1 8583.89,E2 8583.89} C_VEL
LIN {X 0,Y 453.935,Z 808.588,A -85,B 0,C 180,E1 8586.211,E2 8586.211} C_VEL
LIN {X 0,Y 456.93,Z 767.685,A -85,B 0,C 180,E1 8587.705,E2 8587.705} C_VEL
LIN {X 0,Y 457.453,Z 747.509,A -85,B 0,C 180,E1 8588.232,E2 8588.232} C_VEL
LIN {X 0,Y 446.094,Z 724.441,A -85,B 0,C 180,E1 8589.666,E2 8589.666} C_VEL
LIN {X 0,Y 438.561,Z 702.303,A -85,B 0,C 180,E1 8591.067,E2 8591.067} C_VEL
LIN {X 0,Y 432.777,Z 685.03,A -85,B 0,C 180,E1 8593.197,E2 8593.197} C_VEL
LIN {X 0,Y 432.82,Z 685.03,A -85,B 0,C 180,E1 8598.513,E2 8598.513} C_VEL
LIN {X 0,Y 432.816,Z 685.03,A -85,B 0,C 180,E1 8603.649,E2 8603.649} C_VEL
LIN {X 0,Y 432.792,Z 685.03,A -85,B 0,C 180,E1 8608.464,E2 8608.464} C_VEL
LIN {X 0,Y 433.015,Z 685.222,A -85,B 0,C 180,E1 8615.277,E2 8615.277} C_VEL
LIN {X 0,Y 443.818,Z 710.809,A -85,B 0,C 180,E1 8617.627,E2 8617.627} C_VEL
LIN {X 0,Y 446.644,Z 722.13,A -85,B 0,C 180,E1 8618.308,E2 8618.308} C_VEL
LIN {X 0,Y 444.44,Z 773.157,A -85,B 0,C 180,E1 8620.008,E2 8620.008} C_VEL
LIN {X 0,Y 443.072,Z 799.737,A -85,B 0,C 180,E1 8621.634,E2 8621.634} C_VEL
LIN {X 0,Y 441.092,Z 823.978,A -85,B 0,C 180,E1 8623.952,E2 8623.952} C_VEL
LIN {X 0,Y 439.124,Z 844.182,A -85,B 0,C 180,E1 8626.837,E2 8626.837} C_VEL
LIN {X 0,Y 437.455,Z 859.314,A -85,B 0,C 180,E1 8630.065,E2 8630.065} C_VEL
LIN {X 0,Y 436.378,Z 869.555,A -85,B 0,C 180,E1 8633.543,E2 8633.543} C_VEL
LIN {X 0,Y 435.965,Z 873.749,A -85,B 0,C 180,E1 8636.026,E2 8636.026} C_VEL
LIN {X 0,Y 435.67,Z 875.722,A -85,B 0,C 180,E1 8639.996,E2 8639.996} C_VEL
LIN {X 0,Y 435.668,Z 871.881,A -85,B 0,C 180,E1 8643.967,E2 8643.967} C_VEL
LIN {X 0,Y 436.124,Z 861.967,A -85,B 0,C 180,E1 8647.95,E2 8647.95} C_VEL
LIN {X 0,Y 437.168,Z 847.066,A -85,B 0,C 180,E1 8651.442,E2 8651.442} C_VEL
LIN {X 0,Y 438.624,Z 827.984,A -85,B 0,C 180,E1 8654.438,E2 8654.438} C_VEL
LIN {X 0,Y 440.341,Z 803.516,A -85,B 0,C 180,E1 8657.056,E2 8657.056} C_VEL
LIN {X 0,Y 441.882,Z 775.691,A -85,B 0,C 180,E1 8658.989,E2 8658.989} C_VEL
LIN {X 0,Y 442.896,Z 745.717,A -85,B 0,C 180,E1 8660.183,E2 8660.183} C_VEL
LIN {X 0,Y 442.916,Z 715.84,A -85,B 0,C 180,E1 8660.85,E2 8660.85} C_VEL
LIN {X 0,Y 433.169,Z 685.03,A -85,B 0,C 180,E1 8662.106,E2 8662.106} C_VEL
LIN {X 0,Y 432.844,Z 685.03,A -85,B 0,C 180,E1 8669.348,E2 8669.348} C_VEL
LIN {X 0,Y 432.824,Z 685.03,A -85,B 0,C 180,E1 8676.339,E2 8676.339} C_VEL
LIN {X 0,Y 432.806,Z 685.03,A -85,B 0,C 180,E1 8682.923,E2 8682.923} C_VEL
LIN {X 0,Y 432.796,Z 685.03,A -85,B 0,C 180,E1 8688.506,E2 8688.506} C_VEL
LIN {X 0,Y 432.809,Z 685.03,A -85,B 0,C 180,E1 8693.645,E2 8693.645} C_VEL
LIN {X 0,Y 433.057,Z 685.03,A -85,B 0,C 180,E1 8700.618,E2 8700.618} C_VEL
LIN {X 0,Y 446.373,Z 720.645,A -85,B 0,C 180,E1 8702.6,E2 8702.6} C_VEL
LIN {X 0,Y 448.828,Z 732.773,A -85,B 0,C 180,E1 8703.333,E2 8703.333} C_VEL
LIN {X 0,Y 446.633,Z 763.73,A -85,B 0,C 180,E1 8705.147,E2 8705.147} C_VEL
LIN {X 0,Y 443.874,Z 792.231,A -85,B 0,C 180,E1 8707.66,E2 8707.66} C_VEL
LIN {X 0,Y 440.839,Z 817.756,A -85,B 0,C 180,E1 8710.858,E2 8710.858} C_VEL
LIN {X 0,Y 438.248,Z 838.67,A -85,B 0,C 180,E1 8714.569,E2 8714.569} C_VEL
LIN {X 0,Y 436.547,Z 854.039,A -85,B 0,C 180,E1 8718.532,E2 8718.532} C_VEL
LIN {X 0,Y 435.438,Z 865.148,A -85,B 0,C 180,E1 8723.03,E2 8723.03} C_VEL
LIN {X 0,Y 435.134,Z 869.364,A -85,B 0,C 180,E1 8726.02,E2 8726.02} C_VEL
LIN {X 0,Y 435.04,Z 871.343,A -85,B 0,C 180,E1 8729.997,E2 8729.997} C_VEL
LIN {X 0,Y 435.246,Z 868.138,A -85,B 0,C 180,E1 8734.97,E2 8734.97} C_VEL
LIN {X 0,Y 435.978,Z 859.762,A -85,B 0,C 180,E1 8739.363,E2 8739.363} C_VEL
LIN {X 0,Y 437.49,Z 845.654,A -85,B 0,C 180,E1 8743.715,E2 8743.715} C_VEL
LIN {X 0,Y 439.707,Z 827.559,A -85,B 0,C 180,E1 8747.473,E2 8747.473} C_VEL
LIN {X 0,Y 442.541,Z 803.5,A -85,B 0,C 180,E1 8750.978,E2 8750.978} C_VEL
LIN {X 0,Y 445.537,Z 775.924,A -85,B 0,C 180,E1 8753.792,E2 8753.792} C_VEL
LIN {X 0,Y 448.035,Z 744.821,A -85,B 0,C 180,E1 8755.965,E2 8755.965} C_VEL
LIN {X 0,Y 448.306,Z 726.886,A -85,B 0,C 180,E1 8756.892,E2 8756.892} C_VEL
LIN {X 0,Y 436.995,Z 695.694,A -85,B 0,C 180,E1 8758.765,E2 8758.765} C_VEL
LIN {X 0,Y 432.979,Z 685.03,A -85,B 0,C 180,E1 8759.328,E2 8759.328} C_VEL
LIN {X 0,Y 432.852,Z 685.03,A -85,B 0,C 180,E1 8763.901,E2 8763.901} C_VEL
LIN {X 0,Y 432.682,Z 685.03,A -85,B 0,C 180,E1 8769.904,E2 8769.904} C_VEL
LIN {X 0,Y 432.766,Z 685.03,A -85,B 0,C 180,E1 8775.794,E2 8775.794} C_VEL
LIN {X 0,Y 432.795,Z 685.03,A -85,B 0,C 180,E1 8781.137,E2 8781.137} C_VEL
LIN {X 0,Y 432.879,Z 685.03,A -85,B 0,C 180,E1 8786.785,E2 8786.785} C_VEL
LIN {X 0,Y 433.007,Z 685.03,A -85,B 0,C 180,E1 8793.068,E2 8793.068} C_VEL
LIN {X 0,Y 433.304,Z 685.03,A -85,B 0,C 180,E1 8800.099,E2 8800.099} C_VEL
LIN {X 0,Y 433.541,Z 685.03,A -85,B 0,C 180,E1 8805.904,E2 8805.904} C_VEL
LIN {X 0,Y 433.596,Z 685.03,A -85,B 0,C 180,E1 8812.654,E2 8812.654} C_VEL
LIN {X 0,Y 433.812,Z 685.03,A -85,B 0,C 180,E1 8818.011,E2 8818.011} C_VEL
LIN {X 0,Y 433.764,Z 685.03,A -85,B 0,C 180,E1 8823.994,E2 8823.994} C_VEL
LIN {X 0,Y 433.499,Z 685.03,A -85,B 0,C 180,E1 8830.027,E2 8830.027} C_VEL
LIN {X 0,Y 433.307,Z 685.03,A -85,B 0,C 180,E1 8836.18,E2 8836.18} C_VEL
LIN {X 0,Y 433.111,Z 685.03,A -85,B 0,C 180,E1 8842.538,E2 8842.538} C_VEL
LIN {X 0,Y 432.833,Z 685.03,A -85,B 0,C 180,E1 8849.358,E2 8849.358} C_VEL
LIN {X 0,Y 432.819,Z 685.03,A -85,B 0,C 180,E1 8856.35,E2 8856.35} C_VEL
LIN {X 0,Y 432.808,Z 685.03,A -85,B 0,C 180,E1 8862.932,E2 8862.932} C_VEL
LIN {X 0,Y 432.893,Z 685.529,A -85,B 0,C 180,E1 8865.728,E2 8865.728} C_VEL
LIN {X 0,Y 444.253,Z 717.339,A -85,B 0,C 180,E1 8869.081,E2 8869.081} C_VEL
LIN {X 0,Y 459.277,Z 747.785,A -85,B 0,C 180,E1 8871.056,E2 8871.056} C_VEL
LIN {X 0,Y 460.446,Z 750.957,A -85,B 0,C 180,E1 8871.228,E2 8871.228} C_VEL
LIN {X 0,Y 457.875,Z 792.227,A -85,B 0,C 180,E1 8872.423,E2 8872.423} C_VEL
LIN {X 0,Y 454.307,Z 830.278,A -85,B 0,C 180,E1 8874.236,E2 8874.236} C_VEL
LIN {X 0,Y 450.091,Z 866.983,A -85,B 0,C 180,E1 8876.751,E2 8876.751} C_VEL
LIN {X 0,Y 445.578,Z 902.249,A -85,B 0,C 180,E1 8880.049,E2 8880.049} C_VEL
LIN {X 0,Y 440.145,Z 915.303,A -85,B 0,C 180,E1 8881.392,E2 8881.392} C_VEL
